ABB RAPID module: 619bfc00.mod

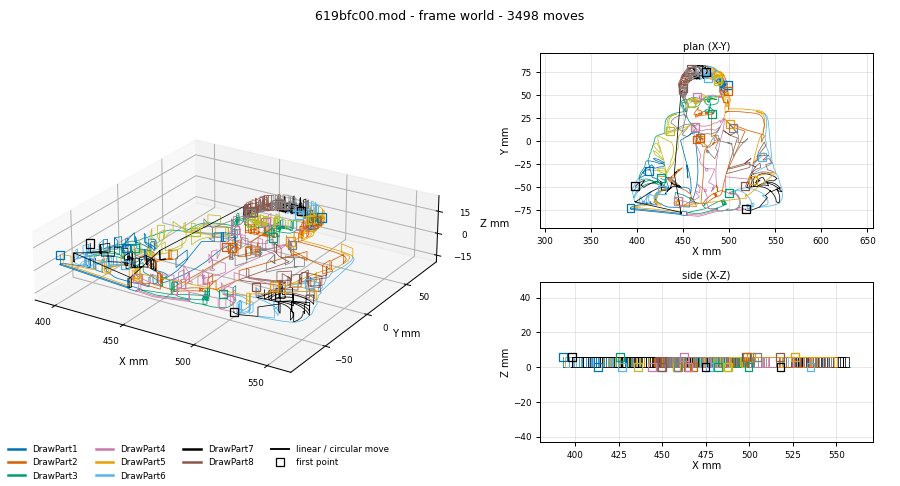
[picture p0: tool path of 619bfc00.mod in frame world, 3498 of 3500 moves have a stored position in this frame; points joined in program order, loops and branches not executed]
MODULE ImageDraw
  ! Generated 2026-10-07 06:22 for ABB GoFa CRB 15000-5/0.95: 344 strokes
  ! Page 250 x 180 mm. Work object wPaper: Z points up, so pen-up is +Z and the tool uses orientation [0,1,0,0].
  PERS tooldata tPen:=[TRUE,[[0,0,120],[1,0,0,0]],[0.3,[0,0,60],[1,0,0,0],0,0,0]];
  PERS wobjdata wPaper:=[FALSE,TRUE,"",[[350,-90,0],[1,0,0,0]],[[0,0,0],[1,0,0,0]]];
  CONST robtarget pOrigin:=[[0,0,0],[0,1,0,0],[0,0,0,0],[9E9,9E9,9E9,9E9,9E9,9E9]];
  CONST jointtarget jHome:=[[0,0,0,0,30,0],[9E9,9E9,9E9,9E9,9E9,9E9]];
  CONST speeddata vTravel:=[250,200,5000,1000];

  PROC DrawImage()
    SingArea\Wrist;
    ConfL\Off;
    ConfJ\Off;
    MoveAbsJ jHome\NoEOffs,vTravel,fine,tPen;
    DrawPart1;
    DrawPart2;
    DrawPart3;
    DrawPart4;
    DrawPart5;
    DrawPart6;
    DrawPart7;
    DrawPart8;
    DrawPart9;
    DrawPart10;
    DrawPart11;
    DrawPart12;
    DrawPart13;
    DrawPart14;
    DrawPart15;
    DrawPart16;
    DrawPart17;
    DrawPart18;
    DrawPart19;
    DrawPart20;
    DrawPart21;
    DrawPart22;
    DrawPart23;
    DrawPart24;
    DrawPart25;
    DrawPart26;
    DrawPart27;
    DrawPart28;
    DrawPart29;
    DrawPart30;
    MoveAbsJ jHome\NoEOffs,vTravel,fine,tPen;
  ENDPROC

  PROC DrawPart1()
    MoveL Offs(pOrigin,42.87,17.43,6.00),vTravel,z5,tPen\WObj:=wPaper;
    MoveL Offs(pOrigin,42.87,17.43,0.00),v60,z0,tPen\WObj:=wPaper;
    MoveL Offs(pOrigin,43.08,16.23,0.00),v40,z0,tPen\WObj:=wPaper;
    MoveL Offs(pOrigin,96.95,10.74,0.00),v40,z0,tPen\WObj:=wPaper;
    MoveL Offs(pOrigin,96.95,10.74,0.00),v40,z0,tPen\WObj:=wPaper;
    MoveL Offs(pOrigin,96.95,12.01,0.00),v40,fine,tPen\WObj:=wPaper;
    MoveL Offs(pOrigin,96.95,12.01,6.00),v60,z5,tPen\WObj:=wPaper;
    MoveL Offs(pOrigin,96.95,10.74,6.00),vTravel,z5,tPen\WObj:=wPaper;
    MoveL Offs(pOrigin,96.95,10.74,0.00),v60,z0,tPen\WObj:=wPaper;
    MoveL Offs(pOrigin,98.22,9.99,0.00),v40,z0,tPen\WObj:=wPaper;
    MoveL Offs(pOrigin,103.43,9.50,0.00),v40,z0,tPen\WObj:=wPaper;
    MoveL Offs(pOrigin,103.54,11.80,0.00),v40,z0,tPen\WObj:=wPaper;
    MoveL Offs(pOrigin,104.39,13.18,0.00),v40,z0,tPen\WObj:=wPaper;
    MoveL Offs(pOrigin,104.39,13.18,0.00),v40,z0,tPen\WObj:=wPaper;
    MoveL Offs(pOrigin,103.96,13.50,0.00),v40,z0,tPen\WObj:=wPaper;
    MoveL Offs(pOrigin,98.44,13.93,0.00),v40,z0,tPen\WObj:=wPaper;
    MoveL Offs(pOrigin,97.27,13.29,0.00),v40,z0,tPen\WObj:=wPaper;
    MoveL Offs(pOrigin,97.27,13.29,0.00),v40,z0,tPen\WObj:=wPaper;
    MoveL Offs(pOrigin,96.91,12.12,0.00),v40,z0,tPen\WObj:=wPaper;
    MoveL Offs(pOrigin,96.10,12.01,0.00),v40,z0,tPen\WObj:=wPaper;
    MoveL Offs(pOrigin,42.87,17.43,0.00),v40,z0,tPen\WObj:=wPaper;
    MoveL Offs(pOrigin,42.87,17.43,0.00),v40,z0,tPen\WObj:=wPaper;
    MoveL Offs(pOrigin,43.08,18.49,0.00),v40,z0,tPen\WObj:=wPaper;
    MoveL Offs(pOrigin,44.04,18.71,0.00),v40,z0,tPen\WObj:=wPaper;
    MoveL Offs(pOrigin,44.04,18.71,0.00),v40,z0,tPen\WObj:=wPaper;
    MoveL Offs(pOrigin,44.36,19.10,0.00),v40,z0,tPen\WObj:=wPaper;
    MoveL Offs(pOrigin,48.29,20.19,0.00),v40,z0,tPen\WObj:=wPaper;
    MoveL Offs(pOrigin,53.81,21.26,0.00),v40,z0,tPen\WObj:=wPaper;
    MoveL Offs(pOrigin,54.66,21.89,0.00),v40,z0,tPen\WObj:=wPaper;
    MoveL Offs(pOrigin,54.66,21.89,0.00),v40,z0,tPen\WObj:=wPaper;
    MoveL Offs(pOrigin,56.36,21.86,0.00),v40,z0,tPen\WObj:=wPaper;
    MoveL Offs(pOrigin,56.26,22.85,0.00),v40,z0,tPen\WObj:=wPaper;
    MoveL Offs(pOrigin,56.26,22.85,0.00),v40,z0,tPen\WObj:=wPaper;
    MoveL Offs(pOrigin,56.19,24.76,0.00),v40,z0,tPen\WObj:=wPaper;
    MoveL Offs(pOrigin,57.11,24.55,0.00),v40,z0,tPen\WObj:=wPaper;
    MoveL Offs(pOrigin,57.11,24.55,0.00),v40,z0,tPen\WObj:=wPaper;
    MoveL Offs(pOrigin,57.74,24.69,0.00),v40,z0,tPen\WObj:=wPaper;
    MoveL Offs(pOrigin,58.17,24.34,0.00),v40,z0,tPen\WObj:=wPaper;
    MoveL Offs(pOrigin,59.12,22.00,0.00),v40,z0,tPen\WObj:=wPaper;
    MoveL Offs(pOrigin,60.61,22.21,0.00),v40,z0,tPen\WObj:=wPaper;
    MoveL Offs(pOrigin,60.51,23.81,0.00),v40,fine,tPen\WObj:=wPaper;
    MoveL Offs(pOrigin,60.51,23.81,6.00),v60,z5,tPen\WObj:=wPaper;
    MoveL Offs(pOrigin,60.72,22.21,6.00),vTravel,z5,tPen\WObj:=wPaper;
    MoveL Offs(pOrigin,60.72,22.21,0.00),v60,z0,tPen\WObj:=wPaper;
    MoveL Offs(pOrigin,61.78,22.42,0.00),v40,fine,tPen\WObj:=wPaper;
    MoveL Offs(pOrigin,61.78,22.42,6.00),v60,z5,tPen\WObj:=wPaper;
    MoveL Offs(pOrigin,63.91,22.64,6.00),vTravel,z5,tPen\WObj:=wPaper;
    MoveL Offs(pOrigin,63.91,22.64,0.00),v60,z0,tPen\WObj:=wPaper;
    MoveL Offs(pOrigin,65.39,22.32,0.00),v40,z0,tPen\WObj:=wPaper;
    MoveL Offs(pOrigin,65.39,22.32,0.00),v40,z0,tPen\WObj:=wPaper;
    MoveL Offs(pOrigin,65.32,23.06,0.00),v40,z0,tPen\WObj:=wPaper;
    MoveL Offs(pOrigin,64.01,24.66,0.00),v40,fine,tPen\WObj:=wPaper;
    MoveL Offs(pOrigin,64.01,24.66,6.00),v60,z5,tPen\WObj:=wPaper;
    MoveL Offs(pOrigin,65.39,22.32,6.00),vTravel,z5,tPen\WObj:=wPaper;
    MoveL Offs(pOrigin,65.39,22.32,0.00),v60,z0,tPen\WObj:=wPaper;
    MoveL Offs(pOrigin,65.82,21.82,0.00),v40,z0,tPen\WObj:=wPaper;
    MoveL Offs(pOrigin,67.09,21.47,0.00),v40,z0,tPen\WObj:=wPaper;
    MoveL Offs(pOrigin,71.34,20.97,0.00),v40,z0,tPen\WObj:=wPaper;
    MoveL Offs(pOrigin,71.27,21.47,0.00),v40,z0,tPen\WObj:=wPaper;
    MoveL Offs(pOrigin,69.43,23.27,0.00),v40,z0,tPen\WObj:=wPaper;
    MoveL Offs(pOrigin,68.47,25.08,0.00),v40,fine,tPen\WObj:=wPaper;
    MoveL Offs(pOrigin,68.47,25.08,6.00),v60,z5,tPen\WObj:=wPaper;
    MoveL Offs(pOrigin,69.86,25.40,6.00),vTravel,z5,tPen\WObj:=wPaper;
    MoveL Offs(pOrigin,69.86,25.40,0.00),v60,z0,tPen\WObj:=wPaper;
    MoveL Offs(pOrigin,69.75,28.06,0.00),v40,z0,tPen\WObj:=wPaper;
    MoveL Offs(pOrigin,69.75,28.06,0.00),v40,z0,tPen\WObj:=wPaper;
    MoveL Offs(pOrigin,70.49,28.02,0.00),v40,z0,tPen\WObj:=wPaper;
    MoveL Offs(pOrigin,70.39,27.21,0.00),v40,z0,tPen\WObj:=wPaper;
    MoveL Offs(pOrigin,70.85,25.51,0.00),v40,z0,tPen\WObj:=wPaper;
    MoveL Offs(pOrigin,71.45,25.29,0.00),v40,z0,tPen\WObj:=wPaper;
    MoveL Offs(pOrigin,71.45,25.29,0.00),v40,z0,tPen\WObj:=wPaper;
    MoveL Offs(pOrigin,72.62,23.59,0.00),v40,z0,tPen\WObj:=wPaper;
    MoveL Offs(pOrigin,74.85,22.81,0.00),v40,z0,tPen\WObj:=wPaper;
    MoveL Offs(pOrigin,75.17,22.32,0.00),v40,z0,tPen\WObj:=wPaper;
    MoveL Offs(pOrigin,75.17,22.32,0.00),v40,z0,tPen\WObj:=wPaper;
    MoveL Offs(pOrigin,76.55,22.14,0.00),v40,z0,tPen\WObj:=wPaper;
    MoveL Offs(pOrigin,77.29,21.29,0.00),v40,z0,tPen\WObj:=wPaper;
    MoveL Offs(pOrigin,81.33,19.31,0.00),v40,z0,tPen\WObj:=wPaper;
    MoveL Offs(pOrigin,84.41,18.60,0.00),v40,z0,tPen\WObj:=wPaper;
    MoveL Offs(pOrigin,94.40,18.39,0.00),v40,z0,tPen\WObj:=wPaper;
    MoveL Offs(pOrigin,97.06,18.60,0.00),v40,z0,tPen\WObj:=wPaper;
    MoveL Offs(pOrigin,99.71,19.34,0.00),v40,z0,tPen\WObj:=wPaper;
    MoveL Offs(pOrigin,99.71,19.34,0.00),v40,z0,tPen\WObj:=wPaper;
    MoveL Offs(pOrigin,100.14,19.02,0.00),v40,z0,tPen\WObj:=wPaper;
    MoveL Offs(pOrigin,106.94,18.71,0.00),v40,fine,tPen\WObj:=wPaper;
    MoveL Offs(pOrigin,106.94,18.71,6.00),v60,z5,tPen\WObj:=wPaper;
    MoveL Offs(pOrigin,106.51,23.59,6.00),vTravel,z5,tPen\WObj:=wPaper;
    MoveL Offs(pOrigin,106.51,23.59,0.00),v60,z0,tPen\WObj:=wPaper;
    MoveL Offs(pOrigin,107.61,24.87,0.00),v40,z0,tPen\WObj:=wPaper;
    MoveL Offs(pOrigin,107.89,26.25,0.00),v40,fine,tPen\WObj:=wPaper;
    MoveL Offs(pOrigin,107.89,26.25,6.00),v60,z5,tPen\WObj:=wPaper;
    MoveL Offs(pOrigin,109.06,27.84,6.00),vTravel,z5,tPen\WObj:=wPaper;
    MoveL Offs(pOrigin,109.06,27.84,0.00),v60,z0,tPen\WObj:=wPaper;
    MoveL Offs(pOrigin,108.00,29.01,0.00),v40,z0,tPen\WObj:=wPaper;
    MoveL Offs(pOrigin,108.53,29.33,0.00),v40,z0,tPen\WObj:=wPaper;
    MoveL Offs(pOrigin,110.12,27.77,0.00),v40,z0,tPen\WObj:=wPaper;
    MoveL Offs(pOrigin,110.66,27.63,0.00),v40,z0,tPen\WObj:=wPaper;
    MoveL Offs(pOrigin,110.66,27.63,0.00),v40,z0,tPen\WObj:=wPaper;
    MoveL Offs(pOrigin,112.14,31.56,0.00),v40,z0,tPen\WObj:=wPaper;
    MoveL Offs(pOrigin,114.27,40.28,0.00),v40,z0,tPen\WObj:=wPaper;
    MoveL Offs(pOrigin,115.01,44.31,0.00),v40,z0,tPen\WObj:=wPaper;
    MoveL Offs(pOrigin,116.07,55.47,0.00),v40,z0,tPen\WObj:=wPaper;
    MoveL Offs(pOrigin,115.86,67.26,0.00),v40,z0,tPen\WObj:=wPaper;
    MoveL Offs(pOrigin,113.74,88.94,0.00),v40,z0,tPen\WObj:=wPaper;
    MoveL Offs(pOrigin,113.74,88.94,0.00),v40,z0,tPen\WObj:=wPaper;
    MoveL Offs(pOrigin,114.27,89.36,0.00),v40,z0,tPen\WObj:=wPaper;
    MoveL Offs(pOrigin,114.48,92.02,0.00),v40,z0,tPen\WObj:=wPaper;
    MoveL Offs(pOrigin,114.48,92.02,0.00),v40,z0,tPen\WObj:=wPaper;
    MoveL Offs(pOrigin,114.91,95.42,0.00),v40,z0,tPen\WObj:=wPaper;
    MoveL Offs(pOrigin,115.76,96.41,0.00),v40,z0,tPen\WObj:=wPaper;
    MoveL Offs(pOrigin,116.29,96.48,0.00),v40,z0,tPen\WObj:=wPaper;
    MoveL Offs(pOrigin,117.24,95.99,0.00),v40,z0,tPen\WObj:=wPaper;
    MoveL Offs(pOrigin,118.73,93.93,0.00),v40,z0,tPen\WObj:=wPaper;
    MoveL Offs(pOrigin,118.52,93.58,0.00),v40,z0,tPen\WObj:=wPaper;
    MoveL Offs(pOrigin,119.09,92.97,0.00),v40,z0,tPen\WObj:=wPaper;
    MoveL Offs(pOrigin,119.47,91.91,0.00),v40,z0,tPen\WObj:=wPaper;
    MoveL Offs(pOrigin,119.26,90.99,0.00),v40,z0,tPen\WObj:=wPaper;
    MoveL Offs(pOrigin,118.52,91.03,0.00),v40,z0,tPen\WObj:=wPaper;
    MoveL Offs(pOrigin,117.85,91.81,0.00),v40,z0,tPen\WObj:=wPaper;
    MoveL Offs(pOrigin,117.56,93.08,0.00),v40,z0,tPen\WObj:=wPaper;
  ENDPROC

  PROC DrawPart2()
    MoveL Offs(pOrigin,117.88,93.54,0.00),v40,z0,tPen\WObj:=wPaper;
    MoveL Offs(pOrigin,118.52,93.58,0.00),v40,z0,tPen\WObj:=wPaper;
    MoveL Offs(pOrigin,118.94,93.08,0.00),v40,z0,tPen\WObj:=wPaper;
    MoveL Offs(pOrigin,118.52,93.51,0.00),v40,z0,tPen\WObj:=wPaper;
    MoveL Offs(pOrigin,118.94,93.08,0.00),v40,fine,tPen\WObj:=wPaper;
    MoveL Offs(pOrigin,118.94,93.08,6.00),v60,z5,tPen\WObj:=wPaper;
    MoveL Offs(pOrigin,120.64,92.97,6.00),vTravel,z5,tPen\WObj:=wPaper;
    MoveL Offs(pOrigin,120.64,92.97,0.00),v60,z0,tPen\WObj:=wPaper;
    MoveL Offs(pOrigin,119.05,95.95,0.00),v40,z0,tPen\WObj:=wPaper;
    MoveL Offs(pOrigin,119.05,95.95,0.00),v40,z0,tPen\WObj:=wPaper;
    MoveL Offs(pOrigin,123.51,94.46,0.00),v40,fine,tPen\WObj:=wPaper;
    MoveL Offs(pOrigin,123.51,94.46,6.00),v60,z5,tPen\WObj:=wPaper;
    MoveL Offs(pOrigin,122.56,92.34,6.00),vTravel,z5,tPen\WObj:=wPaper;
    MoveL Offs(pOrigin,122.56,92.34,0.00),v60,z0,tPen\WObj:=wPaper;
    MoveL Offs(pOrigin,120.64,92.97,0.00),v40,z0,tPen\WObj:=wPaper;
    MoveL Offs(pOrigin,120.64,92.97,0.00),v40,z0,tPen\WObj:=wPaper;
    MoveL Offs(pOrigin,122.41,87.98,0.00),v40,z0,tPen\WObj:=wPaper;
    MoveL Offs(pOrigin,124.68,85.86,0.00),v40,z0,tPen\WObj:=wPaper;
    MoveL Offs(pOrigin,124.89,85.75,0.00),v40,z0,tPen\WObj:=wPaper;
    MoveL Offs(pOrigin,126.49,84.37,0.00),v40,z0,tPen\WObj:=wPaper;
    MoveL Offs(pOrigin,126.49,84.37,0.00),v40,z0,tPen\WObj:=wPaper;
    MoveL Offs(pOrigin,124.47,81.93,0.00),v40,z0,tPen\WObj:=wPaper;
    MoveL Offs(pOrigin,123.58,80.33,0.00),v40,z0,tPen\WObj:=wPaper;
    MoveL Offs(pOrigin,122.66,76.08,0.00),v40,z0,tPen\WObj:=wPaper;
    MoveL Offs(pOrigin,121.71,51.01,0.00),v40,z0,tPen\WObj:=wPaper;
    MoveL Offs(pOrigin,119.37,22.64,0.00),v40,z0,tPen\WObj:=wPaper;
    MoveL Offs(pOrigin,113.21,22.96,0.00),v40,z0,tPen\WObj:=wPaper;
    MoveL Offs(pOrigin,113.21,22.96,0.00),v40,z0,tPen\WObj:=wPaper;
    MoveL Offs(pOrigin,109.06,23.27,0.00),v40,z0,tPen\WObj:=wPaper;
    MoveL Offs(pOrigin,109.06,23.27,0.00),v40,z0,tPen\WObj:=wPaper;
    MoveL Offs(pOrigin,107.26,23.27,0.00),v40,z0,tPen\WObj:=wPaper;
    MoveL Offs(pOrigin,106.51,23.59,0.00),v40,z0,tPen\WObj:=wPaper;
    MoveL Offs(pOrigin,106.51,23.59,0.00),v40,z0,tPen\WObj:=wPaper;
    MoveL Offs(pOrigin,104.92,23.56,0.00),v40,z0,tPen\WObj:=wPaper;
    MoveL Offs(pOrigin,103.64,22.11,0.00),v40,z0,tPen\WObj:=wPaper;
    MoveL Offs(pOrigin,100.67,20.51,0.00),v40,z0,tPen\WObj:=wPaper;
    MoveL Offs(pOrigin,100.67,20.51,0.00),v40,z0,tPen\WObj:=wPaper;
    MoveL Offs(pOrigin,101.09,20.09,0.00),v40,z0,tPen\WObj:=wPaper;
    MoveL Offs(pOrigin,114.48,19.45,0.00),v40,fine,tPen\WObj:=wPaper;
    MoveL Offs(pOrigin,114.48,19.45,6.00),v60,z5,tPen\WObj:=wPaper;
    MoveL Offs(pOrigin,112.99,23.70,6.00),vTravel,z5,tPen\WObj:=wPaper;
    MoveL Offs(pOrigin,112.99,23.70,0.00),v60,z0,tPen\WObj:=wPaper;
    MoveL Offs(pOrigin,112.36,24.76,0.00),v40,z0,tPen\WObj:=wPaper;
    MoveL Offs(pOrigin,112.36,24.76,0.00),v40,z0,tPen\WObj:=wPaper;
    MoveL Offs(pOrigin,110.66,27.63,0.00),v40,fine,tPen\WObj:=wPaper;
    MoveL Offs(pOrigin,110.66,27.63,6.00),v60,z5,tPen\WObj:=wPaper;
    MoveL Offs(pOrigin,110.66,26.36,6.00),vTravel,z5,tPen\WObj:=wPaper;
    MoveL Offs(pOrigin,110.66,26.36,0.00),v60,z0,tPen\WObj:=wPaper;
    MoveL Offs(pOrigin,109.28,27.74,0.00),v40,fine,tPen\WObj:=wPaper;
    MoveL Offs(pOrigin,109.28,27.74,6.00),v60,z5,tPen\WObj:=wPaper;
    MoveL Offs(pOrigin,106.72,28.48,6.00),vTravel,z5,tPen\WObj:=wPaper;
    MoveL Offs(pOrigin,106.72,28.48,0.00),v60,z0,tPen\WObj:=wPaper;
    MoveL Offs(pOrigin,108.53,29.54,0.00),v40,z0,tPen\WObj:=wPaper;
    MoveL Offs(pOrigin,108.74,30.92,0.00),v40,z0,tPen\WObj:=wPaper;
    MoveL Offs(pOrigin,108.00,33.16,0.00),v40,z0,tPen\WObj:=wPaper;
    MoveL Offs(pOrigin,108.00,33.90,0.00),v40,z0,tPen\WObj:=wPaper;
    MoveL Offs(pOrigin,107.89,33.19,0.00),v40,z0,tPen\WObj:=wPaper;
    MoveL Offs(pOrigin,107.15,33.30,0.00),v40,z0,tPen\WObj:=wPaper;
    MoveL Offs(pOrigin,102.58,36.98,0.00),v40,z0,tPen\WObj:=wPaper;
    MoveL Offs(pOrigin,102.58,36.98,0.00),v40,z0,tPen\WObj:=wPaper;
    MoveL Offs(pOrigin,100.24,37.80,0.00),v40,z0,tPen\WObj:=wPaper;
    MoveL Offs(pOrigin,98.33,38.89,0.00),v40,fine,tPen\WObj:=wPaper;
    MoveL Offs(pOrigin,98.33,38.89,6.00),v60,z5,tPen\WObj:=wPaper;
    MoveL Offs(pOrigin,97.80,40.28,6.00),vTravel,z5,tPen\WObj:=wPaper;
    MoveL Offs(pOrigin,97.80,40.28,0.00),v60,z0,tPen\WObj:=wPaper;
    MoveL Offs(pOrigin,95.04,42.22,0.00),v40,z0,tPen\WObj:=wPaper;
    MoveL Offs(pOrigin,94.65,43.14,0.00),v40,z0,tPen\WObj:=wPaper;
    MoveL Offs(pOrigin,94.19,43.36,0.00),v40,z0,tPen\WObj:=wPaper;
    MoveL Offs(pOrigin,94.19,43.36,0.00),v40,z0,tPen\WObj:=wPaper;
    MoveL Offs(pOrigin,91.21,46.33,0.00),v40,z0,tPen\WObj:=wPaper;
    MoveL Offs(pOrigin,90.47,46.86,0.00),v40,z0,tPen\WObj:=wPaper;
    MoveL Offs(pOrigin,90.93,46.47,0.00),v40,z0,tPen\WObj:=wPaper;
    MoveL Offs(pOrigin,86.36,50.37,0.00),v40,z0,tPen\WObj:=wPaper;
    MoveL Offs(pOrigin,95.46,59.72,0.00),v40,fine,tPen\WObj:=wPaper;
    MoveL Offs(pOrigin,95.46,59.72,6.00),v60,z5,tPen\WObj:=wPaper;
    MoveL Offs(pOrigin,94.29,58.66,6.00),vTravel,z5,tPen\WObj:=wPaper;
    MoveL Offs(pOrigin,94.29,58.66,0.00),v60,z0,tPen\WObj:=wPaper;
    MoveL Offs(pOrigin,94.82,59.19,0.00),v40,z0,tPen\WObj:=wPaper;
    MoveL Offs(pOrigin,94.29,58.66,0.00),v40,z0,tPen\WObj:=wPaper;
    MoveL Offs(pOrigin,95.25,58.12,0.00),v40,z0,tPen\WObj:=wPaper;
    MoveL Offs(pOrigin,96.42,59.29,0.00),v40,z0,tPen\WObj:=wPaper;
    MoveL Offs(pOrigin,95.25,58.12,0.00),v40,fine,tPen\WObj:=wPaper;
    MoveL Offs(pOrigin,95.25,58.12,6.00),v60,z5,tPen\WObj:=wPaper;
    MoveL Offs(pOrigin,98.97,61.31,6.00),vTravel,z5,tPen\WObj:=wPaper;
    MoveL Offs(pOrigin,98.97,61.31,0.00),v60,z0,tPen\WObj:=wPaper;
    MoveL Offs(pOrigin,93.66,56.32,0.00),v40,z0,tPen\WObj:=wPaper;
    MoveL Offs(pOrigin,91.18,52.81,0.00),v40,z0,tPen\WObj:=wPaper;
    MoveL Offs(pOrigin,89.62,49.84,0.00),v40,fine,tPen\WObj:=wPaper;
    MoveL Offs(pOrigin,89.62,49.84,6.00),v60,z5,tPen\WObj:=wPaper;
    MoveL Offs(pOrigin,87.07,51.33,6.00),vTravel,z5,tPen\WObj:=wPaper;
    MoveL Offs(pOrigin,87.07,51.33,0.00),v60,z0,tPen\WObj:=wPaper;
    MoveL Offs(pOrigin,87.49,51.75,0.00),v40,z0,tPen\WObj:=wPaper;
    MoveL Offs(pOrigin,87.07,51.33,0.00),v40,z0,tPen\WObj:=wPaper;
    MoveL Offs(pOrigin,86.32,50.47,0.00),v40,z0,tPen\WObj:=wPaper;
    MoveL Offs(pOrigin,84.84,50.79,0.00),v40,z0,tPen\WObj:=wPaper;
    MoveL Offs(pOrigin,84.84,50.79,0.00),v40,z0,tPen\WObj:=wPaper;
    MoveL Offs(pOrigin,83.24,49.20,0.00),v40,z0,tPen\WObj:=wPaper;
    MoveL Offs(pOrigin,83.24,49.20,0.00),v40,z0,tPen\WObj:=wPaper;
    MoveL Offs(pOrigin,83.99,48.03,0.00),v40,z0,tPen\WObj:=wPaper;
    MoveL Offs(pOrigin,90.36,42.22,0.00),v40,z0,tPen\WObj:=wPaper;
    MoveL Offs(pOrigin,90.79,41.48,0.00),v40,z0,tPen\WObj:=wPaper;
    MoveL Offs(pOrigin,93.09,41.02,0.00),v40,z0,tPen\WObj:=wPaper;
    MoveL Offs(pOrigin,93.09,41.55,0.00),v40,z0,tPen\WObj:=wPaper;
    MoveL Offs(pOrigin,88.45,45.69,0.00),v40,z0,tPen\WObj:=wPaper;
    MoveL Offs(pOrigin,87.92,46.01,0.00),v40,z0,tPen\WObj:=wPaper;
    MoveL Offs(pOrigin,88.17,45.84,0.00),v40,z0,tPen\WObj:=wPaper;
    MoveL Offs(pOrigin,84.62,48.88,0.00),v40,fine,tPen\WObj:=wPaper;
    MoveL Offs(pOrigin,84.62,48.88,6.00),v60,z5,tPen\WObj:=wPaper;
    MoveL Offs(pOrigin,83.24,49.20,6.00),vTravel,z5,tPen\WObj:=wPaper;
    MoveL Offs(pOrigin,83.24,49.20,0.00),v60,z0,tPen\WObj:=wPaper;
    MoveL Offs(pOrigin,82.89,49.52,0.00),v40,z0,tPen\WObj:=wPaper;
    MoveL Offs(pOrigin,82.82,50.26,0.00),v40,z0,tPen\WObj:=wPaper;
    MoveL Offs(pOrigin,82.82,50.26,0.00),v40,z0,tPen\WObj:=wPaper;
    MoveL Offs(pOrigin,81.83,51.11,0.00),v40,z0,tPen\WObj:=wPaper;
    MoveL Offs(pOrigin,81.44,53.45,0.00),v40,z0,tPen\WObj:=wPaper;
    MoveL Offs(pOrigin,81.44,53.45,0.00),v40,z0,tPen\WObj:=wPaper;
    MoveL Offs(pOrigin,80.27,52.25,0.00),v40,z0,tPen\WObj:=wPaper;
    MoveL Offs(pOrigin,78.99,51.96,0.00),v40,z0,tPen\WObj:=wPaper;
    MoveL Offs(pOrigin,73.26,52.28,0.00),v40,fine,tPen\WObj:=wPaper;
    MoveL Offs(pOrigin,73.26,52.28,6.00),v60,z5,tPen\WObj:=wPaper;
  ENDPROC

  PROC DrawPart3()
    MoveL Offs(pOrigin,75.70,49.84,6.00),vTravel,z5,tPen\WObj:=wPaper;
    MoveL Offs(pOrigin,75.70,49.84,0.00),v60,z0,tPen\WObj:=wPaper;
    MoveL Offs(pOrigin,79.10,48.14,0.00),v40,z0,tPen\WObj:=wPaper;
    MoveL Offs(pOrigin,80.48,48.67,0.00),v40,z0,tPen\WObj:=wPaper;
    MoveL Offs(pOrigin,80.48,48.67,0.00),v40,z0,tPen\WObj:=wPaper;
    MoveL Offs(pOrigin,80.38,44.53,0.00),v40,z0,tPen\WObj:=wPaper;
    MoveL Offs(pOrigin,79.21,41.12,0.00),v40,z0,tPen\WObj:=wPaper;
    MoveL Offs(pOrigin,75.06,42.36,0.00),v40,z0,tPen\WObj:=wPaper;
    MoveL Offs(pOrigin,72.41,43.53,0.00),v40,z0,tPen\WObj:=wPaper;
    MoveL Offs(pOrigin,69.01,46.15,0.00),v40,z0,tPen\WObj:=wPaper;
    MoveL Offs(pOrigin,65.39,47.71,0.00),v40,z0,tPen\WObj:=wPaper;
    MoveL Offs(pOrigin,65.39,47.71,0.00),v40,z0,tPen\WObj:=wPaper;
    MoveL Offs(pOrigin,65.07,47.29,0.00),v40,z0,tPen\WObj:=wPaper;
    MoveL Offs(pOrigin,62.42,47.39,0.00),v40,z0,tPen\WObj:=wPaper;
    MoveL Offs(pOrigin,60.40,46.90,0.00),v40,z0,tPen\WObj:=wPaper;
    MoveL Offs(pOrigin,58.06,45.84,0.00),v40,z0,tPen\WObj:=wPaper;
    MoveL Offs(pOrigin,55.94,44.31,0.00),v40,z0,tPen\WObj:=wPaper;
    MoveL Offs(pOrigin,52.29,39.96,0.00),v40,z0,tPen\WObj:=wPaper;
    MoveL Offs(pOrigin,50.59,36.77,0.00),v40,z0,tPen\WObj:=wPaper;
    MoveL Offs(pOrigin,49.99,34.86,0.00),v40,z0,tPen\WObj:=wPaper;
    MoveL Offs(pOrigin,49.99,34.86,0.00),v40,z0,tPen\WObj:=wPaper;
    MoveL Offs(pOrigin,51.90,36.34,0.00),v40,z0,tPen\WObj:=wPaper;
    MoveL Offs(pOrigin,55.94,41.02,0.00),v40,z0,tPen\WObj:=wPaper;
    MoveL Offs(pOrigin,57.74,42.44,0.00),v40,z0,tPen\WObj:=wPaper;
    MoveL Offs(pOrigin,61.25,43.89,0.00),v40,z0,tPen\WObj:=wPaper;
    MoveL Offs(pOrigin,64.12,44.21,0.00),v40,z0,tPen\WObj:=wPaper;
    MoveL Offs(pOrigin,64.12,44.21,0.00),v40,z0,tPen\WObj:=wPaper;
    MoveL Offs(pOrigin,67.09,44.31,0.00),v40,z0,tPen\WObj:=wPaper;
    MoveL Offs(pOrigin,71.77,43.78,0.00),v40,fine,tPen\WObj:=wPaper;
    MoveL Offs(pOrigin,71.77,43.78,6.00),v60,z5,tPen\WObj:=wPaper;
    MoveL Offs(pOrigin,69.86,45.27,6.00),vTravel,z5,tPen\WObj:=wPaper;
    MoveL Offs(pOrigin,69.86,45.27,0.00),v60,z0,tPen\WObj:=wPaper;
    MoveL Offs(pOrigin,69.32,45.16,0.00),v40,z0,tPen\WObj:=wPaper;
    MoveL Offs(pOrigin,67.94,45.87,0.00),v40,z0,tPen\WObj:=wPaper;
    MoveL Offs(pOrigin,67.62,46.65,0.00),v40,fine,tPen\WObj:=wPaper;
    MoveL Offs(pOrigin,67.62,46.65,6.00),v60,z5,tPen\WObj:=wPaper;
    MoveL Offs(pOrigin,65.39,47.71,6.00),vTravel,z5,tPen\WObj:=wPaper;
    MoveL Offs(pOrigin,65.39,47.71,0.00),v60,z0,tPen\WObj:=wPaper;
    MoveL Offs(pOrigin,63.91,48.46,0.00),v40,z0,tPen\WObj:=wPaper;
    MoveL Offs(pOrigin,60.51,49.20,0.00),v40,z0,tPen\WObj:=wPaper;
    MoveL Offs(pOrigin,56.26,48.99,0.00),v40,z0,tPen\WObj:=wPaper;
    MoveL Offs(pOrigin,53.07,47.92,0.00),v40,fine,tPen\WObj:=wPaper;
    MoveL Offs(pOrigin,53.07,47.92,6.00),v60,z5,tPen\WObj:=wPaper;
    MoveL Offs(pOrigin,52.01,49.84,6.00),vTravel,z5,tPen\WObj:=wPaper;
    MoveL Offs(pOrigin,52.01,49.84,0.00),v60,z0,tPen\WObj:=wPaper;
    MoveL Offs(pOrigin,52.86,53.34,0.00),v40,z0,tPen\WObj:=wPaper;
    MoveL Offs(pOrigin,54.10,56.53,0.00),v40,z0,tPen\WObj:=wPaper;
    MoveL Offs(pOrigin,58.10,61.95,0.00),v40,z0,tPen\WObj:=wPaper;
    MoveL Offs(pOrigin,59.41,67.69,0.00),v40,z0,tPen\WObj:=wPaper;
    MoveL Offs(pOrigin,60.51,68.79,0.00),v40,z0,tPen\WObj:=wPaper;
    MoveL Offs(pOrigin,61.89,69.07,0.00),v40,z0,tPen\WObj:=wPaper;
    MoveL Offs(pOrigin,61.89,69.07,0.00),v40,z0,tPen\WObj:=wPaper;
    MoveL Offs(pOrigin,62.03,70.56,0.00),v40,z0,tPen\WObj:=wPaper;
    MoveL Offs(pOrigin,63.48,72.79,0.00),v40,z0,tPen\WObj:=wPaper;
    MoveL Offs(pOrigin,63.66,76.19,0.00),v40,z0,tPen\WObj:=wPaper;
    MoveL Offs(pOrigin,64.90,77.68,0.00),v40,z0,tPen\WObj:=wPaper;
    MoveL Offs(pOrigin,65.18,78.53,0.00),v40,z0,tPen\WObj:=wPaper;
    MoveL Offs(pOrigin,65.25,81.18,0.00),v40,z0,tPen\WObj:=wPaper;
    MoveL Offs(pOrigin,66.78,82.99,0.00),v40,z0,tPen\WObj:=wPaper;
    MoveL Offs(pOrigin,66.88,85.43,0.00),v40,z0,tPen\WObj:=wPaper;
    MoveL Offs(pOrigin,67.59,86.39,0.00),v40,z0,tPen\WObj:=wPaper;
    MoveL Offs(pOrigin,68.47,89.15,0.00),v40,z0,tPen\WObj:=wPaper;
    MoveL Offs(pOrigin,69.50,93.72,0.00),v40,z0,tPen\WObj:=wPaper;
    MoveL Offs(pOrigin,71.03,95.84,0.00),v40,z0,tPen\WObj:=wPaper;
    MoveL Offs(pOrigin,72.51,96.38,0.00),v40,z0,tPen\WObj:=wPaper;
    MoveL Offs(pOrigin,72.51,96.38,0.00),v40,z0,tPen\WObj:=wPaper;
    MoveL Offs(pOrigin,75.06,97.44,0.00),v40,z0,tPen\WObj:=wPaper;
    MoveL Offs(pOrigin,79.84,98.78,0.00),v40,z0,tPen\WObj:=wPaper;
    MoveL Offs(pOrigin,80.16,99.14,0.00),v40,z0,tPen\WObj:=wPaper;
    MoveL Offs(pOrigin,80.16,99.14,0.00),v40,z0,tPen\WObj:=wPaper;
    MoveL Offs(pOrigin,80.16,105.83,0.00),v40,z0,tPen\WObj:=wPaper;
    MoveL Offs(pOrigin,80.59,110.82,0.00),v40,z0,tPen\WObj:=wPaper;
    MoveL Offs(pOrigin,81.40,113.59,0.00),v40,z0,tPen\WObj:=wPaper;
    MoveL Offs(pOrigin,82.93,116.03,0.00),v40,z0,tPen\WObj:=wPaper;
    MoveL Offs(pOrigin,85.37,118.09,0.00),v40,z0,tPen\WObj:=wPaper;
    MoveL Offs(pOrigin,89.30,119.89,0.00),v40,z0,tPen\WObj:=wPaper;
    MoveL Offs(pOrigin,93.02,120.92,0.00),v40,z0,tPen\WObj:=wPaper;
    MoveL Offs(pOrigin,100.88,122.30,0.00),v40,z0,tPen\WObj:=wPaper;
    MoveL Offs(pOrigin,100.88,122.30,0.00),v40,z0,tPen\WObj:=wPaper;
    MoveL Offs(pOrigin,100.17,124.85,0.00),v40,z0,tPen\WObj:=wPaper;
    MoveL Offs(pOrigin,98.37,127.82,0.00),v40,z0,tPen\WObj:=wPaper;
    MoveL Offs(pOrigin,97.69,130.06,0.00),v40,z0,tPen\WObj:=wPaper;
    MoveL Offs(pOrigin,98.08,133.03,0.00),v40,z0,tPen\WObj:=wPaper;
    MoveL Offs(pOrigin,98.86,134.09,0.00),v40,z0,tPen\WObj:=wPaper;
    MoveL Offs(pOrigin,100.03,134.73,0.00),v40,z0,tPen\WObj:=wPaper;
    MoveL Offs(pOrigin,100.14,135.48,0.00),v40,z0,tPen\WObj:=wPaper;
    MoveL Offs(pOrigin,100.14,134.73,0.00),v40,z0,tPen\WObj:=wPaper;
    MoveL Offs(pOrigin,101.41,134.41,0.00),v40,z0,tPen\WObj:=wPaper;
    MoveL Offs(pOrigin,101.41,134.41,0.00),v40,z0,tPen\WObj:=wPaper;
    MoveL Offs(pOrigin,101.55,133.14,0.00),v40,z0,tPen\WObj:=wPaper;
    MoveL Offs(pOrigin,102.05,132.61,0.00),v40,z0,tPen\WObj:=wPaper;
    MoveL Offs(pOrigin,102.58,132.18,0.00),v40,z0,tPen\WObj:=wPaper;
    MoveL Offs(pOrigin,102.37,131.44,0.00),v40,z0,tPen\WObj:=wPaper;
    MoveL Offs(pOrigin,100.56,132.36,0.00),v40,z0,tPen\WObj:=wPaper;
    MoveL Offs(pOrigin,99.54,132.39,0.00),v40,z0,tPen\WObj:=wPaper;
    MoveL Offs(pOrigin,99.07,129.84,0.00),v40,z0,tPen\WObj:=wPaper;
    MoveL Offs(pOrigin,100.03,127.61,0.00),v40,fine,tPen\WObj:=wPaper;
    MoveL Offs(pOrigin,100.03,127.61,6.00),v60,z5,tPen\WObj:=wPaper;
    MoveL Offs(pOrigin,100.67,129.21,6.00),vTravel,z5,tPen\WObj:=wPaper;
    MoveL Offs(pOrigin,100.67,129.21,0.00),v60,z0,tPen\WObj:=wPaper;
    MoveL Offs(pOrigin,100.78,126.44,0.00),v40,z0,tPen\WObj:=wPaper;
    MoveL Offs(pOrigin,102.47,122.30,0.00),v40,z0,tPen\WObj:=wPaper;
    MoveL Offs(pOrigin,103.32,122.62,0.00),v40,z0,tPen\WObj:=wPaper;
    MoveL Offs(pOrigin,103.22,123.68,0.00),v40,fine,tPen\WObj:=wPaper;
    MoveL Offs(pOrigin,103.22,123.68,6.00),v60,z5,tPen\WObj:=wPaper;
    MoveL Offs(pOrigin,103.54,121.13,6.00),vTravel,z5,tPen\WObj:=wPaper;
    MoveL Offs(pOrigin,103.54,121.13,0.00),v60,z0,tPen\WObj:=wPaper;
    MoveL Offs(pOrigin,104.18,116.35,0.00),v40,z0,tPen\WObj:=wPaper;
    MoveL Offs(pOrigin,104.18,116.35,0.00),v40,z0,tPen\WObj:=wPaper;
    MoveL Offs(pOrigin,106.19,112.31,0.00),v40,z0,tPen\WObj:=wPaper;
    MoveL Offs(pOrigin,108.64,109.27,0.00),v40,z0,tPen\WObj:=wPaper;
    MoveL Offs(pOrigin,110.02,108.49,0.00),v40,z0,tPen\WObj:=wPaper;
    MoveL Offs(pOrigin,110.02,108.49,0.00),v40,z0,tPen\WObj:=wPaper;
    MoveL Offs(pOrigin,113.31,107.11,0.00),v40,fine,tPen\WObj:=wPaper;
    MoveL Offs(pOrigin,113.31,107.11,6.00),v60,z5,tPen\WObj:=wPaper;
    MoveL Offs(pOrigin,111.72,106.26,6.00),vTravel,z5,tPen\WObj:=wPaper;
    MoveL Offs(pOrigin,111.72,106.26,0.00),v60,z0,tPen\WObj:=wPaper;
    MoveL Offs(pOrigin,110.97,107.00,0.00),v40,z0,tPen\WObj:=wPaper;
    MoveL Offs(pOrigin,111.72,106.26,0.00),v40,fine,tPen\WObj:=wPaper;
    MoveL Offs(pOrigin,111.72,106.26,6.00),v60,z5,tPen\WObj:=wPaper;
  ENDPROC

  PROC DrawPart4()
    MoveL Offs(pOrigin,112.68,105.30,6.00),vTravel,z5,tPen\WObj:=wPaper;
    MoveL Offs(pOrigin,112.68,105.30,0.00),v60,z0,tPen\WObj:=wPaper;
    MoveL Offs(pOrigin,111.82,106.15,0.00),v40,z0,tPen\WObj:=wPaper;
    MoveL Offs(pOrigin,112.68,105.30,0.00),v40,fine,tPen\WObj:=wPaper;
    MoveL Offs(pOrigin,112.68,105.30,6.00),v60,z5,tPen\WObj:=wPaper;
    MoveL Offs(pOrigin,113.53,104.34,6.00),vTravel,z5,tPen\WObj:=wPaper;
    MoveL Offs(pOrigin,113.53,104.34,0.00),v60,z0,tPen\WObj:=wPaper;
    MoveL Offs(pOrigin,110.83,107.28,0.00),v40,z0,tPen\WObj:=wPaper;
    MoveL Offs(pOrigin,110.27,107.53,0.00),v40,z0,tPen\WObj:=wPaper;
    MoveL Offs(pOrigin,110.02,108.49,0.00),v40,z0,tPen\WObj:=wPaper;
    MoveL Offs(pOrigin,110.23,107.43,0.00),v40,z0,tPen\WObj:=wPaper;
    MoveL Offs(pOrigin,111.19,100.41,0.00),v40,z0,tPen\WObj:=wPaper;
    MoveL Offs(pOrigin,111.19,100.41,0.00),v40,z0,tPen\WObj:=wPaper;
    MoveL Offs(pOrigin,112.46,95.42,0.00),v40,z0,tPen\WObj:=wPaper;
    MoveL Offs(pOrigin,113.42,89.26,0.00),v40,z0,tPen\WObj:=wPaper;
    MoveL Offs(pOrigin,113.74,88.94,0.00),v40,fine,tPen\WObj:=wPaper;
    MoveL Offs(pOrigin,113.74,88.94,6.00),v60,z5,tPen\WObj:=wPaper;
    MoveL Offs(pOrigin,114.06,86.28,6.00),vTravel,z5,tPen\WObj:=wPaper;
    MoveL Offs(pOrigin,114.06,86.28,0.00),v60,z0,tPen\WObj:=wPaper;
    MoveL Offs(pOrigin,114.66,85.86,0.00),v40,z0,tPen\WObj:=wPaper;
    MoveL Offs(pOrigin,119.37,74.28,0.00),v40,fine,tPen\WObj:=wPaper;
    MoveL Offs(pOrigin,119.37,74.28,6.00),v60,z5,tPen\WObj:=wPaper;
    MoveL Offs(pOrigin,117.78,70.34,6.00),vTravel,z5,tPen\WObj:=wPaper;
    MoveL Offs(pOrigin,117.78,70.34,0.00),v60,z0,tPen\WObj:=wPaper;
    MoveL Offs(pOrigin,118.62,66.31,0.00),v40,fine,tPen\WObj:=wPaper;
    MoveL Offs(pOrigin,118.62,66.31,6.00),v60,z5,tPen\WObj:=wPaper;
    MoveL Offs(pOrigin,124.86,60.39,6.00),vTravel,z5,tPen\WObj:=wPaper;
    MoveL Offs(pOrigin,124.86,60.39,0.00),v60,z0,tPen\WObj:=wPaper;
    MoveL Offs(pOrigin,125.85,60.57,0.00),v40,z0,tPen\WObj:=wPaper;
    MoveL Offs(pOrigin,126.59,60.14,0.00),v40,z0,tPen\WObj:=wPaper;
    MoveL Offs(pOrigin,127.02,59.08,0.00),v40,z0,tPen\WObj:=wPaper;
    MoveL Offs(pOrigin,126.59,58.02,0.00),v40,z0,tPen\WObj:=wPaper;
    MoveL Offs(pOrigin,125.21,57.70,0.00),v40,z0,tPen\WObj:=wPaper;
    MoveL Offs(pOrigin,124.47,58.12,0.00),v40,z0,tPen\WObj:=wPaper;
    MoveL Offs(pOrigin,124.15,59.51,0.00),v40,z0,tPen\WObj:=wPaper;
    MoveL Offs(pOrigin,124.86,60.39,0.00),v40,fine,tPen\WObj:=wPaper;
    MoveL Offs(pOrigin,124.86,60.39,6.00),v60,z5,tPen\WObj:=wPaper;
    MoveL Offs(pOrigin,134.35,60.04,6.00),vTravel,z5,tPen\WObj:=wPaper;
    MoveL Offs(pOrigin,134.35,60.04,0.00),v60,z0,tPen\WObj:=wPaper;
    MoveL Offs(pOrigin,131.09,52.17,0.00),v40,z0,tPen\WObj:=wPaper;
    MoveL Offs(pOrigin,127.55,45.48,0.00),v40,fine,tPen\WObj:=wPaper;
    MoveL Offs(pOrigin,127.55,45.48,6.00),v60,z5,tPen\WObj:=wPaper;
    MoveL Offs(pOrigin,133.93,42.19,6.00),vTravel,z5,tPen\WObj:=wPaper;
    MoveL Offs(pOrigin,133.93,42.19,0.00),v60,z0,tPen\WObj:=wPaper;
    MoveL Offs(pOrigin,131.69,39.32,0.00),v40,fine,tPen\WObj:=wPaper;
    MoveL Offs(pOrigin,131.69,39.32,6.00),v60,z5,tPen\WObj:=wPaper;
    MoveL Offs(pOrigin,132.65,38.26,6.00),vTravel,z5,tPen\WObj:=wPaper;
    MoveL Offs(pOrigin,132.65,38.26,0.00),v60,z0,tPen\WObj:=wPaper;
    MoveL Offs(pOrigin,132.97,38.58,0.00),v40,z0,tPen\WObj:=wPaper;
    MoveL Offs(pOrigin,132.65,38.26,0.00),v40,z0,tPen\WObj:=wPaper;
    MoveL Offs(pOrigin,133.29,39.00,0.00),v40,z0,tPen\WObj:=wPaper;
    MoveL Offs(pOrigin,133.61,39.32,0.00),v40,z0,tPen\WObj:=wPaper;
    MoveL Offs(pOrigin,133.29,39.00,0.00),v40,fine,tPen\WObj:=wPaper;
    MoveL Offs(pOrigin,133.29,39.00,6.00),v60,z5,tPen\WObj:=wPaper;
    MoveL Offs(pOrigin,130.42,35.81,6.00),vTravel,z5,tPen\WObj:=wPaper;
    MoveL Offs(pOrigin,130.42,35.81,0.00),v60,z0,tPen\WObj:=wPaper;
    MoveL Offs(pOrigin,136.37,42.72,0.00),v40,z0,tPen\WObj:=wPaper;
    MoveL Offs(pOrigin,136.37,42.72,0.00),v40,z0,tPen\WObj:=wPaper;
    MoveL Offs(pOrigin,135.62,51.22,0.00),v40,z0,tPen\WObj:=wPaper;
    MoveL Offs(pOrigin,135.62,59.83,0.00),v40,z0,tPen\WObj:=wPaper;
    MoveL Offs(pOrigin,136.48,69.28,0.00),v40,z0,tPen\WObj:=wPaper;
    MoveL Offs(pOrigin,137.86,78.84,0.00),v40,z0,tPen\WObj:=wPaper;
    MoveL Offs(pOrigin,137.86,78.84,0.00),v40,z0,tPen\WObj:=wPaper;
    MoveL Offs(pOrigin,140.19,90.21,0.00),v40,z0,tPen\WObj:=wPaper;
    MoveL Offs(pOrigin,143.38,102.01,0.00),v40,z0,tPen\WObj:=wPaper;
    MoveL Offs(pOrigin,143.38,102.01,0.00),v40,z0,tPen\WObj:=wPaper;
    MoveL Offs(pOrigin,144.55,109.23,0.00),v40,z0,tPen\WObj:=wPaper;
    MoveL Offs(pOrigin,144.55,113.16,0.00),v40,z0,tPen\WObj:=wPaper;
    MoveL Offs(pOrigin,144.12,113.91,0.00),v40,z0,tPen\WObj:=wPaper;
    MoveL Offs(pOrigin,144.02,114.76,0.00),v40,z0,tPen\WObj:=wPaper;
    MoveL Offs(pOrigin,143.27,114.33,0.00),v40,z0,tPen\WObj:=wPaper;
    MoveL Offs(pOrigin,140.51,110.40,0.00),v40,fine,tPen\WObj:=wPaper;
    MoveL Offs(pOrigin,140.51,110.40,6.00),v60,z5,tPen\WObj:=wPaper;
    MoveL Offs(pOrigin,140.19,113.06,6.00),vTravel,z5,tPen\WObj:=wPaper;
    MoveL Offs(pOrigin,140.19,113.06,0.00),v60,z0,tPen\WObj:=wPaper;
    MoveL Offs(pOrigin,136.90,110.08,0.00),v40,fine,tPen\WObj:=wPaper;
    MoveL Offs(pOrigin,136.90,110.08,6.00),v60,z5,tPen\WObj:=wPaper;
    MoveL Offs(pOrigin,133.61,109.97,6.00),vTravel,z5,tPen\WObj:=wPaper;
    MoveL Offs(pOrigin,133.61,109.97,0.00),v60,z0,tPen\WObj:=wPaper;
    MoveL Offs(pOrigin,130.21,107.81,0.00),v40,z0,tPen\WObj:=wPaper;
    MoveL Offs(pOrigin,127.23,107.00,0.00),v40,z0,tPen\WObj:=wPaper;
    MoveL Offs(pOrigin,123.51,106.47,0.00),v40,z0,tPen\WObj:=wPaper;
    MoveL Offs(pOrigin,118.84,106.79,0.00),v40,z0,tPen\WObj:=wPaper;
    MoveL Offs(pOrigin,116.61,107.71,0.00),v40,z0,tPen\WObj:=wPaper;
    MoveL Offs(pOrigin,114.59,109.02,0.00),v40,fine,tPen\WObj:=wPaper;
    MoveL Offs(pOrigin,114.59,109.02,6.00),v60,z5,tPen\WObj:=wPaper;
    MoveL Offs(pOrigin,113.53,104.34,6.00),vTravel,z5,tPen\WObj:=wPaper;
    MoveL Offs(pOrigin,113.53,104.34,0.00),v60,z0,tPen\WObj:=wPaper;
    MoveL Offs(pOrigin,117.03,102.40,0.00),v40,z0,tPen\WObj:=wPaper;
    MoveL Offs(pOrigin,119.69,101.37,0.00),v40,fine,tPen\WObj:=wPaper;
    MoveL Offs(pOrigin,119.69,101.37,6.00),v60,z5,tPen\WObj:=wPaper;
    MoveL Offs(pOrigin,122.45,101.90,6.00),vTravel,z5,tPen\WObj:=wPaper;
    MoveL Offs(pOrigin,122.45,101.90,0.00),v60,z0,tPen\WObj:=wPaper;
    MoveL Offs(pOrigin,125.53,103.07,0.00),v40,z0,tPen\WObj:=wPaper;
    MoveL Offs(pOrigin,129.14,102.75,0.00),v40,z0,tPen\WObj:=wPaper;
    MoveL Offs(pOrigin,131.06,102.96,0.00),v40,fine,tPen\WObj:=wPaper;
    MoveL Offs(pOrigin,131.06,102.96,6.00),v60,z5,tPen\WObj:=wPaper;
    MoveL Offs(pOrigin,134.88,102.11,6.00),vTravel,z5,tPen\WObj:=wPaper;
    MoveL Offs(pOrigin,134.88,102.11,0.00),v60,z0,tPen\WObj:=wPaper;
    MoveL Offs(pOrigin,140.19,105.83,0.00),v40,z0,tPen\WObj:=wPaper;
    MoveL Offs(pOrigin,140.19,105.83,0.00),v40,z0,tPen\WObj:=wPaper;
    MoveL Offs(pOrigin,142.99,111.25,0.00),v40,z0,tPen\WObj:=wPaper;
    MoveL Offs(pOrigin,144.12,114.12,0.00),v40,z0,tPen\WObj:=wPaper;
    MoveL Offs(pOrigin,144.12,115.07,0.00),v40,fine,tPen\WObj:=wPaper;
    MoveL Offs(pOrigin,144.12,115.07,6.00),v60,z5,tPen\WObj:=wPaper;
    MoveL Offs(pOrigin,148.06,111.14,6.00),vTravel,z5,tPen\WObj:=wPaper;
    MoveL Offs(pOrigin,148.06,111.14,0.00),v60,z0,tPen\WObj:=wPaper;
    MoveL Offs(pOrigin,147.21,111.99,0.00),v40,z0,tPen\WObj:=wPaper;
    MoveL Offs(pOrigin,148.06,111.14,0.00),v40,fine,tPen\WObj:=wPaper;
    MoveL Offs(pOrigin,148.06,111.14,6.00),v60,z5,tPen\WObj:=wPaper;
    MoveL Offs(pOrigin,148.91,110.29,6.00),vTravel,z5,tPen\WObj:=wPaper;
    MoveL Offs(pOrigin,148.91,110.29,0.00),v60,z0,tPen\WObj:=wPaper;
    MoveL Offs(pOrigin,148.16,111.04,0.00),v40,z0,tPen\WObj:=wPaper;
    MoveL Offs(pOrigin,148.91,110.29,0.00),v40,fine,tPen\WObj:=wPaper;
    MoveL Offs(pOrigin,148.91,110.29,6.00),v60,z5,tPen\WObj:=wPaper;
    MoveL Offs(pOrigin,149.86,109.34,6.00),vTravel,z5,tPen\WObj:=wPaper;
    MoveL Offs(pOrigin,149.86,109.34,0.00),v60,z0,tPen\WObj:=wPaper;
    MoveL Offs(pOrigin,149.01,110.19,0.00),v40,z0,tPen\WObj:=wPaper;
    MoveL Offs(pOrigin,149.86,109.34,0.00),v40,fine,tPen\WObj:=wPaper;
    MoveL Offs(pOrigin,149.86,109.34,6.00),v60,z5,tPen\WObj:=wPaper;
  ENDPROC

  PROC DrawPart5()
    MoveL Offs(pOrigin,151.03,108.70,6.00),vTravel,z5,tPen\WObj:=wPaper;
    MoveL Offs(pOrigin,151.03,108.70,0.00),v60,z0,tPen\WObj:=wPaper;
    MoveL Offs(pOrigin,150.18,109.12,0.00),v40,z0,tPen\WObj:=wPaper;
    MoveL Offs(pOrigin,145.29,114.44,0.00),v40,z0,tPen\WObj:=wPaper;
    MoveL Offs(pOrigin,144.16,115.18,0.00),v40,z0,tPen\WObj:=wPaper;
    MoveL Offs(pOrigin,145.40,119.32,0.00),v40,z0,tPen\WObj:=wPaper;
    MoveL Offs(pOrigin,145.72,121.77,0.00),v40,z0,tPen\WObj:=wPaper;
    MoveL Offs(pOrigin,145.72,121.77,0.00),v40,z0,tPen\WObj:=wPaper;
    MoveL Offs(pOrigin,145.29,126.34,0.00),v40,z0,tPen\WObj:=wPaper;
    MoveL Offs(pOrigin,145.40,127.51,0.00),v40,z0,tPen\WObj:=wPaper;
    MoveL Offs(pOrigin,145.93,128.57,0.00),v40,z0,tPen\WObj:=wPaper;
    MoveL Offs(pOrigin,145.93,128.57,0.00),v40,z0,tPen\WObj:=wPaper;
    MoveL Offs(pOrigin,146.14,130.59,0.00),v40,z0,tPen\WObj:=wPaper;
    MoveL Offs(pOrigin,144.87,132.82,0.00),v40,z0,tPen\WObj:=wPaper;
    MoveL Offs(pOrigin,145.40,132.93,0.00),v40,z0,tPen\WObj:=wPaper;
    MoveL Offs(pOrigin,146.46,131.54,0.00),v40,fine,tPen\WObj:=wPaper;
    MoveL Offs(pOrigin,146.46,131.54,6.00),v60,z5,tPen\WObj:=wPaper;
    MoveL Offs(pOrigin,147.42,130.69,6.00),vTravel,z5,tPen\WObj:=wPaper;
    MoveL Offs(pOrigin,147.42,130.69,0.00),v60,z0,tPen\WObj:=wPaper;
    MoveL Offs(pOrigin,146.89,129.21,0.00),v40,z0,tPen\WObj:=wPaper;
    MoveL Offs(pOrigin,145.93,128.57,0.00),v40,fine,tPen\WObj:=wPaper;
    MoveL Offs(pOrigin,145.93,128.57,6.00),v60,z5,tPen\WObj:=wPaper;
    MoveL Offs(pOrigin,147.63,127.40,6.00),vTravel,z5,tPen\WObj:=wPaper;
    MoveL Offs(pOrigin,147.63,127.40,0.00),v60,z0,tPen\WObj:=wPaper;
    MoveL Offs(pOrigin,148.52,128.78,0.00),v40,z0,tPen\WObj:=wPaper;
    MoveL Offs(pOrigin,149.86,133.88,0.00),v40,z0,tPen\WObj:=wPaper;
    MoveL Offs(pOrigin,149.86,135.69,0.00),v40,z0,tPen\WObj:=wPaper;
    MoveL Offs(pOrigin,148.91,137.78,0.00),v40,z0,tPen\WObj:=wPaper;
    MoveL Offs(pOrigin,148.16,138.13,0.00),v40,z0,tPen\WObj:=wPaper;
    MoveL Offs(pOrigin,146.78,137.39,0.00),v40,z0,tPen\WObj:=wPaper;
    MoveL Offs(pOrigin,145.58,135.58,0.00),v40,z0,tPen\WObj:=wPaper;
    MoveL Offs(pOrigin,144.98,133.35,0.00),v40,z0,tPen\WObj:=wPaper;
    MoveL Offs(pOrigin,144.98,133.35,0.00),v40,z0,tPen\WObj:=wPaper;
    MoveL Offs(pOrigin,144.66,132.85,0.00),v40,z0,tPen\WObj:=wPaper;
    MoveL Offs(pOrigin,143.91,133.46,0.00),v40,z0,tPen\WObj:=wPaper;
    MoveL Offs(pOrigin,143.91,133.46,0.00),v40,z0,tPen\WObj:=wPaper;
    MoveL Offs(pOrigin,143.81,134.52,0.00),v40,z0,tPen\WObj:=wPaper;
    MoveL Offs(pOrigin,144.12,135.37,0.00),v40,z0,tPen\WObj:=wPaper;
    MoveL Offs(pOrigin,143.81,134.73,0.00),v40,z0,tPen\WObj:=wPaper;
    MoveL Offs(pOrigin,143.17,135.05,0.00),v40,z0,tPen\WObj:=wPaper;
    MoveL Offs(pOrigin,142.96,135.90,0.00),v40,z0,tPen\WObj:=wPaper;
    MoveL Offs(pOrigin,142.96,135.90,0.00),v40,z0,tPen\WObj:=wPaper;
    MoveL Offs(pOrigin,144.02,136.11,0.00),v40,z0,tPen\WObj:=wPaper;
    MoveL Offs(pOrigin,143.91,136.54,0.00),v40,z0,tPen\WObj:=wPaper;
    MoveL Offs(pOrigin,144.02,137.81,0.00),v40,z0,tPen\WObj:=wPaper;
    MoveL Offs(pOrigin,144.02,137.81,0.00),v40,z0,tPen\WObj:=wPaper;
    MoveL Offs(pOrigin,142.53,137.78,0.00),v40,z0,tPen\WObj:=wPaper;
    MoveL Offs(pOrigin,142.74,136.64,0.00),v40,z0,tPen\WObj:=wPaper;
    MoveL Offs(pOrigin,142.74,136.64,0.00),v40,z0,tPen\WObj:=wPaper;
    MoveL Offs(pOrigin,143.91,136.54,0.00),v40,fine,tPen\WObj:=wPaper;
    MoveL Offs(pOrigin,143.91,136.54,6.00),v60,z5,tPen\WObj:=wPaper;
    MoveL Offs(pOrigin,144.44,137.92,6.00),vTravel,z5,tPen\WObj:=wPaper;
    MoveL Offs(pOrigin,144.44,137.92,0.00),v60,z0,tPen\WObj:=wPaper;
    MoveL Offs(pOrigin,144.66,138.63,0.00),v40,z0,tPen\WObj:=wPaper;
    MoveL Offs(pOrigin,146.57,139.51,0.00),v40,z0,tPen\WObj:=wPaper;
    MoveL Offs(pOrigin,147.10,140.36,0.00),v40,z0,tPen\WObj:=wPaper;
    MoveL Offs(pOrigin,147.31,140.36,0.00),v40,z0,tPen\WObj:=wPaper;
    MoveL Offs(pOrigin,147.74,140.04,0.00),v40,z0,tPen\WObj:=wPaper;
    MoveL Offs(pOrigin,148.91,140.15,0.00),v40,z0,tPen\WObj:=wPaper;
    MoveL Offs(pOrigin,148.91,140.15,0.00),v40,z0,tPen\WObj:=wPaper;
    MoveL Offs(pOrigin,149.33,140.47,0.00),v40,z0,tPen\WObj:=wPaper;
    MoveL Offs(pOrigin,149.01,141.96,0.00),v40,z0,tPen\WObj:=wPaper;
    MoveL Offs(pOrigin,148.80,141.96,0.00),v40,z0,tPen\WObj:=wPaper;
    MoveL Offs(pOrigin,149.12,143.34,0.00),v40,z0,tPen\WObj:=wPaper;
    MoveL Offs(pOrigin,148.27,143.23,0.00),v40,z0,tPen\WObj:=wPaper;
    MoveL Offs(pOrigin,147.21,141.53,0.00),v40,z0,tPen\WObj:=wPaper;
    MoveL Offs(pOrigin,147.21,141.53,0.00),v40,z0,tPen\WObj:=wPaper;
    MoveL Offs(pOrigin,144.66,141.21,0.00),v40,z0,tPen\WObj:=wPaper;
    MoveL Offs(pOrigin,144.66,141.21,0.00),v40,z0,tPen\WObj:=wPaper;
    MoveL Offs(pOrigin,145.40,140.57,0.00),v40,z0,tPen\WObj:=wPaper;
    MoveL Offs(pOrigin,145.40,140.57,0.00),v40,z0,tPen\WObj:=wPaper;
    MoveL Offs(pOrigin,147.21,140.43,0.00),v40,z0,tPen\WObj:=wPaper;
    MoveL Offs(pOrigin,147.42,141.11,0.00),v40,z0,tPen\WObj:=wPaper;
    MoveL Offs(pOrigin,148.27,141.00,0.00),v40,z0,tPen\WObj:=wPaper;
    MoveL Offs(pOrigin,148.80,141.96,0.00),v40,z0,tPen\WObj:=wPaper;
    MoveL Offs(pOrigin,148.80,141.96,0.00),v40,z0,tPen\WObj:=wPaper;
    MoveL Offs(pOrigin,147.84,142.06,0.00),v40,z0,tPen\WObj:=wPaper;
    MoveL Offs(pOrigin,148.27,141.00,0.00),v40,z0,tPen\WObj:=wPaper;
    MoveL Offs(pOrigin,148.91,140.36,0.00),v40,z0,tPen\WObj:=wPaper;
    MoveL Offs(pOrigin,149.33,140.26,0.00),v40,z0,tPen\WObj:=wPaper;
    MoveL Offs(pOrigin,150.75,137.49,0.00),v40,z0,tPen\WObj:=wPaper;
    MoveL Offs(pOrigin,151.35,134.52,0.00),v40,z0,tPen\WObj:=wPaper;
    MoveL Offs(pOrigin,149.33,125.38,0.00),v40,z0,tPen\WObj:=wPaper;
    MoveL Offs(pOrigin,149.33,125.38,0.00),v40,z0,tPen\WObj:=wPaper;
    MoveL Offs(pOrigin,163.99,125.17,0.00),v40,z0,tPen\WObj:=wPaper;
    MoveL Offs(pOrigin,179.08,123.79,0.00),v40,z0,tPen\WObj:=wPaper;
    MoveL Offs(pOrigin,183.23,123.04,0.00),v40,z0,tPen\WObj:=wPaper;
    MoveL Offs(pOrigin,186.31,122.02,0.00),v40,z0,tPen\WObj:=wPaper;
    MoveL Offs(pOrigin,187.90,120.99,0.00),v40,z0,tPen\WObj:=wPaper;
    MoveL Offs(pOrigin,188.64,119.75,0.00),v40,fine,tPen\WObj:=wPaper;
    MoveL Offs(pOrigin,188.64,119.75,6.00),v60,z5,tPen\WObj:=wPaper;
    MoveL Offs(pOrigin,179.19,122.30,6.00),vTravel,z5,tPen\WObj:=wPaper;
    MoveL Offs(pOrigin,179.19,122.30,0.00),v60,z0,tPen\WObj:=wPaper;
    MoveL Offs(pOrigin,181.52,122.09,0.00),v40,z0,tPen\WObj:=wPaper;
    MoveL Offs(pOrigin,183.65,121.49,0.00),v40,z0,tPen\WObj:=wPaper;
    MoveL Offs(pOrigin,185.46,120.56,0.00),v40,z0,tPen\WObj:=wPaper;
    MoveL Offs(pOrigin,186.62,119.43,0.00),v40,z0,tPen\WObj:=wPaper;
    MoveL Offs(pOrigin,187.51,117.84,0.00),v40,z0,tPen\WObj:=wPaper;
    MoveL Offs(pOrigin,188.22,115.29,0.00),v40,z0,tPen\WObj:=wPaper;
    MoveL Offs(pOrigin,188.54,112.42,0.00),v40,z0,tPen\WObj:=wPaper;
    MoveL Offs(pOrigin,188.32,109.02,0.00),v40,z0,tPen\WObj:=wPaper;
    MoveL Offs(pOrigin,188.32,109.02,0.00),v40,z0,tPen\WObj:=wPaper;
    MoveL Offs(pOrigin,188.11,105.62,0.00),v40,z0,tPen\WObj:=wPaper;
    MoveL Offs(pOrigin,186.52,97.44,0.00),v40,z0,tPen\WObj:=wPaper;
    MoveL Offs(pOrigin,186.52,97.44,0.00),v40,z0,tPen\WObj:=wPaper;
    MoveL Offs(pOrigin,185.35,97.44,0.00),v40,z0,tPen\WObj:=wPaper;
    MoveL Offs(pOrigin,185.35,97.44,0.00),v40,z0,tPen\WObj:=wPaper;
    MoveL Offs(pOrigin,183.51,94.14,0.00),v40,z0,tPen\WObj:=wPaper;
    MoveL Offs(pOrigin,181.42,87.98,0.00),v40,z0,tPen\WObj:=wPaper;
    MoveL Offs(pOrigin,177.81,74.38,0.00),v40,z0,tPen\WObj:=wPaper;
    MoveL Offs(pOrigin,176.32,66.84,0.00),v40,z0,tPen\WObj:=wPaper;
    MoveL Offs(pOrigin,176.32,66.84,0.00),v40,z0,tPen\WObj:=wPaper;
    MoveL Offs(pOrigin,176.96,67.26,0.00),v40,z0,tPen\WObj:=wPaper;
    MoveL Offs(pOrigin,178.34,69.39,0.00),v40,z0,tPen\WObj:=wPaper;
    MoveL Offs(pOrigin,181.42,73.00,0.00),v40,z0,tPen\WObj:=wPaper;
    MoveL Offs(pOrigin,183.97,75.34,0.00),v40,z0,tPen\WObj:=wPaper;
    MoveL Offs(pOrigin,187.48,77.78,0.00),v40,fine,tPen\WObj:=wPaper;
    MoveL Offs(pOrigin,187.48,77.78,6.00),v60,z5,tPen\WObj:=wPaper;
    MoveL Offs(pOrigin,188.32,74.49,6.00),vTravel,z5,tPen\WObj:=wPaper;
    MoveL Offs(pOrigin,188.32,74.49,0.00),v60,z0,tPen\WObj:=wPaper;
  ENDPROC

  PROC DrawPart6()
    MoveL Offs(pOrigin,185.14,73.25,0.00),v40,z0,tPen\WObj:=wPaper;
    MoveL Offs(pOrigin,183.23,72.04,0.00),v40,z0,tPen\WObj:=wPaper;
    MoveL Offs(pOrigin,178.98,67.90,0.00),v40,z0,tPen\WObj:=wPaper;
    MoveL Offs(pOrigin,176.64,64.29,0.00),v40,z0,tPen\WObj:=wPaper;
    MoveL Offs(pOrigin,175.93,63.76,0.00),v40,z0,tPen\WObj:=wPaper;
    MoveL Offs(pOrigin,174.62,58.66,0.00),v40,z0,tPen\WObj:=wPaper;
    MoveL Offs(pOrigin,174.51,56.96,0.00),v40,z0,tPen\WObj:=wPaper;
    MoveL Offs(pOrigin,174.51,56.96,0.00),v40,z0,tPen\WObj:=wPaper;
    MoveL Offs(pOrigin,174.09,55.36,0.00),v40,z0,tPen\WObj:=wPaper;
    MoveL Offs(pOrigin,174.09,55.36,0.00),v40,z0,tPen\WObj:=wPaper;
    MoveL Offs(pOrigin,174.30,53.24,0.00),v40,z0,tPen\WObj:=wPaper;
    MoveL Offs(pOrigin,178.76,56.74,0.00),v40,z0,tPen\WObj:=wPaper;
    MoveL Offs(pOrigin,183.23,59.44,0.00),v40,z0,tPen\WObj:=wPaper;
    MoveL Offs(pOrigin,189.81,62.73,0.00),v40,z0,tPen\WObj:=wPaper;
    MoveL Offs(pOrigin,193.64,64.07,0.00),v40,fine,tPen\WObj:=wPaper;
    MoveL Offs(pOrigin,193.64,64.07,6.00),v60,z5,tPen\WObj:=wPaper;
    MoveL Offs(pOrigin,195.44,66.41,6.00),vTravel,z5,tPen\WObj:=wPaper;
    MoveL Offs(pOrigin,195.44,66.41,0.00),v60,z0,tPen\WObj:=wPaper;
    MoveL Offs(pOrigin,194.70,72.36,0.00),v40,z0,tPen\WObj:=wPaper;
    MoveL Offs(pOrigin,192.89,74.70,0.00),v40,z0,tPen\WObj:=wPaper;
    MoveL Offs(pOrigin,192.89,74.70,0.00),v40,z0,tPen\WObj:=wPaper;
    MoveL Offs(pOrigin,193.11,77.25,0.00),v40,z0,tPen\WObj:=wPaper;
    MoveL Offs(pOrigin,189.88,85.22,0.00),v40,z0,tPen\WObj:=wPaper;
    MoveL Offs(pOrigin,190.45,88.09,0.00),v40,z0,tPen\WObj:=wPaper;
    MoveL Offs(pOrigin,189.39,91.17,0.00),v40,z0,tPen\WObj:=wPaper;
    MoveL Offs(pOrigin,188.75,94.68,0.00),v40,z0,tPen\WObj:=wPaper;
    MoveL Offs(pOrigin,189.28,95.31,0.00),v40,z0,tPen\WObj:=wPaper;
    MoveL Offs(pOrigin,190.56,106.79,0.00),v40,z0,tPen\WObj:=wPaper;
    MoveL Offs(pOrigin,190.34,113.80,0.00),v40,z0,tPen\WObj:=wPaper;
    MoveL Offs(pOrigin,189.92,116.35,0.00),v40,z0,tPen\WObj:=wPaper;
    MoveL Offs(pOrigin,188.68,119.43,0.00),v40,z0,tPen\WObj:=wPaper;
    MoveL Offs(pOrigin,189.07,119.96,0.00),v40,z0,tPen\WObj:=wPaper;
    MoveL Offs(pOrigin,191.02,117.20,0.00),v40,z0,tPen\WObj:=wPaper;
    MoveL Offs(pOrigin,192.47,111.78,0.00),v40,z0,tPen\WObj:=wPaper;
    MoveL Offs(pOrigin,196.72,66.41,0.00),v40,z0,tPen\WObj:=wPaper;
    MoveL Offs(pOrigin,196.72,66.41,0.00),v40,z0,tPen\WObj:=wPaper;
    MoveL Offs(pOrigin,197.85,65.67,0.00),v40,z0,tPen\WObj:=wPaper;
    MoveL Offs(pOrigin,198.17,61.10,0.00),v40,z0,tPen\WObj:=wPaper;
    MoveL Offs(pOrigin,199.84,58.44,0.00),v40,z0,tPen\WObj:=wPaper;
    MoveL Offs(pOrigin,200.51,55.58,0.00),v40,z0,tPen\WObj:=wPaper;
    MoveL Offs(pOrigin,203.24,51.33,0.00),v40,z0,tPen\WObj:=wPaper;
    MoveL Offs(pOrigin,205.01,44.74,0.00),v40,z0,tPen\WObj:=wPaper;
    MoveL Offs(pOrigin,207.13,39.21,0.00),v40,z0,tPen\WObj:=wPaper;
    MoveL Offs(pOrigin,207.56,37.41,0.00),v40,z0,tPen\WObj:=wPaper;
    MoveL Offs(pOrigin,207.34,34.86,0.00),v40,z0,tPen\WObj:=wPaper;
    MoveL Offs(pOrigin,207.88,31.35,0.00),v40,z0,tPen\WObj:=wPaper;
    MoveL Offs(pOrigin,207.34,27.63,0.00),v40,z0,tPen\WObj:=wPaper;
    MoveL Offs(pOrigin,205.54,24.12,0.00),v40,z0,tPen\WObj:=wPaper;
    MoveL Offs(pOrigin,203.73,22.71,0.00),v40,z0,tPen\WObj:=wPaper;
    MoveL Offs(pOrigin,201.93,21.86,0.00),v40,z0,tPen\WObj:=wPaper;
    MoveL Offs(pOrigin,198.63,20.83,0.00),v40,z0,tPen\WObj:=wPaper;
    MoveL Offs(pOrigin,192.89,19.66,0.00),v40,z0,tPen\WObj:=wPaper;
    MoveL Offs(pOrigin,183.12,18.39,0.00),v40,z0,tPen\WObj:=wPaper;
    MoveL Offs(pOrigin,182.80,18.60,0.00),v40,z0,tPen\WObj:=wPaper;
    MoveL Offs(pOrigin,182.80,18.60,0.00),v40,z0,tPen\WObj:=wPaper;
    MoveL Offs(pOrigin,183.33,19.27,0.00),v40,z0,tPen\WObj:=wPaper;
    MoveL Offs(pOrigin,192.04,21.79,0.00),v40,fine,tPen\WObj:=wPaper;
    MoveL Offs(pOrigin,192.04,21.79,6.00),v60,z5,tPen\WObj:=wPaper;
    MoveL Offs(pOrigin,192.15,25.72,6.00),vTravel,z5,tPen\WObj:=wPaper;
    MoveL Offs(pOrigin,192.15,25.72,0.00),v60,z0,tPen\WObj:=wPaper;
    MoveL Offs(pOrigin,188.86,28.91,0.00),v40,z0,tPen\WObj:=wPaper;
    MoveL Offs(pOrigin,188.64,29.01,0.00),v40,z0,tPen\WObj:=wPaper;
    MoveL Offs(pOrigin,185.77,31.46,0.00),v40,fine,tPen\WObj:=wPaper;
    MoveL Offs(pOrigin,185.77,31.46,6.00),v60,z5,tPen\WObj:=wPaper;
    MoveL Offs(pOrigin,188.96,31.35,6.00),vTravel,z5,tPen\WObj:=wPaper;
    MoveL Offs(pOrigin,188.96,31.35,0.00),v60,z0,tPen\WObj:=wPaper;
    MoveL Offs(pOrigin,185.46,34.04,0.00),v40,z0,tPen\WObj:=wPaper;
    MoveL Offs(pOrigin,180.78,36.49,0.00),v40,z0,tPen\WObj:=wPaper;
    MoveL Offs(pOrigin,174.83,38.36,0.00),v40,z0,tPen\WObj:=wPaper;
    MoveL Offs(pOrigin,170.90,38.89,0.00),v40,fine,tPen\WObj:=wPaper;
    MoveL Offs(pOrigin,170.90,38.89,6.00),v60,z5,tPen\WObj:=wPaper;
    MoveL Offs(pOrigin,168.99,39.85,6.00),vTravel,z5,tPen\WObj:=wPaper;
    MoveL Offs(pOrigin,168.99,39.85,0.00),v60,z0,tPen\WObj:=wPaper;
    MoveL Offs(pOrigin,159.64,38.04,0.00),v40,z0,tPen\WObj:=wPaper;
    MoveL Offs(pOrigin,156.98,37.02,0.00),v40,z0,tPen\WObj:=wPaper;
    MoveL Offs(pOrigin,156.56,36.34,0.00),v40,z0,tPen\WObj:=wPaper;
    MoveL Offs(pOrigin,156.56,36.34,0.00),v40,z0,tPen\WObj:=wPaper;
    MoveL Offs(pOrigin,160.49,36.56,0.00),v40,z0,tPen\WObj:=wPaper;
    MoveL Offs(pOrigin,164.21,35.32,0.00),v40,z0,tPen\WObj:=wPaper;
    MoveL Offs(pOrigin,167.71,33.05,0.00),v40,z0,tPen\WObj:=wPaper;
    MoveL Offs(pOrigin,171.22,29.33,0.00),v40,z0,tPen\WObj:=wPaper;
    MoveL Offs(pOrigin,173.91,24.98,0.00),v40,z0,tPen\WObj:=wPaper;
    MoveL Offs(pOrigin,175.15,21.36,0.00),v40,z0,tPen\WObj:=wPaper;
    MoveL Offs(pOrigin,174.65,18.28,0.00),v40,z0,tPen\WObj:=wPaper;
    MoveL Offs(pOrigin,173.56,16.58,0.00),v40,z0,tPen\WObj:=wPaper;
    MoveL Offs(pOrigin,172.28,15.62,0.00),v40,z0,tPen\WObj:=wPaper;
    MoveL Offs(pOrigin,171.96,14.99,0.00),v40,fine,tPen\WObj:=wPaper;
    MoveL Offs(pOrigin,171.96,14.99,6.00),v60,z5,tPen\WObj:=wPaper;
    MoveL Offs(pOrigin,171.22,16.65,6.00),vTravel,z5,tPen\WObj:=wPaper;
    MoveL Offs(pOrigin,171.22,16.65,0.00),v60,z0,tPen\WObj:=wPaper;
    MoveL Offs(pOrigin,171.71,17.01,0.00),v40,z0,tPen\WObj:=wPaper;
    MoveL Offs(pOrigin,171.61,17.54,0.00),v40,z0,tPen\WObj:=wPaper;
    MoveL Offs(pOrigin,170.26,17.25,0.00),v40,z0,tPen\WObj:=wPaper;
    MoveL Offs(pOrigin,169.84,16.58,0.00),v40,z0,tPen\WObj:=wPaper;
    MoveL Offs(pOrigin,171.22,16.65,0.00),v40,z0,tPen\WObj:=wPaper;
    MoveL Offs(pOrigin,171.75,17.54,0.00),v40,z0,tPen\WObj:=wPaper;
    MoveL Offs(pOrigin,173.27,19.34,0.00),v40,z0,tPen\WObj:=wPaper;
    MoveL Offs(pOrigin,174.41,22.85,0.00),v40,fine,tPen\WObj:=wPaper;
    MoveL Offs(pOrigin,174.41,22.85,6.00),v60,z5,tPen\WObj:=wPaper;
    MoveL Offs(pOrigin,177.27,22.21,6.00),vTravel,z5,tPen\WObj:=wPaper;
    MoveL Offs(pOrigin,177.27,22.21,0.00),v60,z0,tPen\WObj:=wPaper;
    MoveL Offs(pOrigin,176.43,19.24,0.00),v40,fine,tPen\WObj:=wPaper;
    MoveL Offs(pOrigin,176.43,19.24,6.00),v60,z5,tPen\WObj:=wPaper;
    MoveL Offs(pOrigin,170.94,19.66,6.00),vTravel,z5,tPen\WObj:=wPaper;
    MoveL Offs(pOrigin,170.94,19.66,0.00),v60,z0,tPen\WObj:=wPaper;
    MoveL Offs(pOrigin,171.22,21.04,0.00),v40,z0,tPen\WObj:=wPaper;
    MoveL Offs(pOrigin,170.79,21.75,0.00),v40,z0,tPen\WObj:=wPaper;
    MoveL Offs(pOrigin,169.73,21.82,0.00),v40,z0,tPen\WObj:=wPaper;
    MoveL Offs(pOrigin,168.85,20.94,0.00),v40,z0,tPen\WObj:=wPaper;
    MoveL Offs(pOrigin,168.56,19.88,0.00),v40,z0,tPen\WObj:=wPaper;
    MoveL Offs(pOrigin,169.31,18.99,0.00),v40,z0,tPen\WObj:=wPaper;
    MoveL Offs(pOrigin,170.26,19.06,0.00),v40,z0,tPen\WObj:=wPaper;
    MoveL Offs(pOrigin,170.94,19.66,0.00),v40,fine,tPen\WObj:=wPaper;
    MoveL Offs(pOrigin,170.94,19.66,6.00),v60,z5,tPen\WObj:=wPaper;
    MoveL Offs(pOrigin,169.09,20.19,6.00),vTravel,z5,tPen\WObj:=wPaper;
    MoveL Offs(pOrigin,169.09,20.19,0.00),v60,z0,tPen\WObj:=wPaper;
    MoveL Offs(pOrigin,169.62,21.26,0.00),v40,fine,tPen\WObj:=wPaper;
    MoveL Offs(pOrigin,169.62,21.26,6.00),v60,z5,tPen\WObj:=wPaper;
    MoveL Offs(pOrigin,169.73,16.79,6.00),vTravel,z5,tPen\WObj:=wPaper;
    MoveL Offs(pOrigin,169.73,16.79,0.00),v60,z0,tPen\WObj:=wPaper;
  ENDPROC

  PROC DrawPart7()
    MoveL Offs(pOrigin,167.93,16.58,0.00),v40,z0,tPen\WObj:=wPaper;
    MoveL Offs(pOrigin,167.50,16.26,0.00),v40,z0,tPen\WObj:=wPaper;
    MoveL Offs(pOrigin,167.50,16.26,0.00),v40,z0,tPen\WObj:=wPaper;
    MoveL Offs(pOrigin,167.93,15.70,0.00),v40,z0,tPen\WObj:=wPaper;
    MoveL Offs(pOrigin,169.62,15.09,0.00),v40,z0,tPen\WObj:=wPaper;
    MoveL Offs(pOrigin,172.71,14.88,0.00),v40,z0,tPen\WObj:=wPaper;
    MoveL Offs(pOrigin,182.80,18.60,0.00),v40,fine,tPen\WObj:=wPaper;
    MoveL Offs(pOrigin,182.80,18.60,6.00),v60,z5,tPen\WObj:=wPaper;
    MoveL Offs(pOrigin,191.51,28.91,6.00),vTravel,z5,tPen\WObj:=wPaper;
    MoveL Offs(pOrigin,191.51,28.91,0.00),v60,z0,tPen\WObj:=wPaper;
    MoveL Offs(pOrigin,189.18,31.24,0.00),v40,fine,tPen\WObj:=wPaper;
    MoveL Offs(pOrigin,189.18,31.24,6.00),v60,z5,tPen\WObj:=wPaper;
    MoveL Offs(pOrigin,194.81,36.03,6.00),vTravel,z5,tPen\WObj:=wPaper;
    MoveL Offs(pOrigin,194.81,36.03,0.00),v60,z0,tPen\WObj:=wPaper;
    MoveL Offs(pOrigin,194.49,36.34,0.00),v40,z0,tPen\WObj:=wPaper;
    MoveL Offs(pOrigin,194.81,36.03,0.00),v40,z0,tPen\WObj:=wPaper;
    MoveL Offs(pOrigin,195.44,35.49,0.00),v40,z0,tPen\WObj:=wPaper;
    MoveL Offs(pOrigin,191.94,38.29,0.00),v40,z0,tPen\WObj:=wPaper;
    MoveL Offs(pOrigin,188.96,39.78,0.00),v40,z0,tPen\WObj:=wPaper;
    MoveL Offs(pOrigin,186.41,40.49,0.00),v40,z0,tPen\WObj:=wPaper;
    MoveL Offs(pOrigin,180.89,41.12,0.00),v40,fine,tPen\WObj:=wPaper;
    MoveL Offs(pOrigin,180.89,41.12,6.00),v60,z5,tPen\WObj:=wPaper;
    MoveL Offs(pOrigin,183.54,42.29,6.00),vTravel,z5,tPen\WObj:=wPaper;
    MoveL Offs(pOrigin,183.54,42.29,0.00),v60,z0,tPen\WObj:=wPaper;
    MoveL Offs(pOrigin,188.11,42.72,0.00),v40,z0,tPen\WObj:=wPaper;
    MoveL Offs(pOrigin,192.89,41.76,0.00),v40,fine,tPen\WObj:=wPaper;
    MoveL Offs(pOrigin,192.89,41.76,6.00),v60,z5,tPen\WObj:=wPaper;
    MoveL Offs(pOrigin,190.98,45.06,6.00),vTravel,z5,tPen\WObj:=wPaper;
    MoveL Offs(pOrigin,190.98,45.06,0.00),v60,z0,tPen\WObj:=wPaper;
    MoveL Offs(pOrigin,197.25,42.97,0.00),v40,z0,tPen\WObj:=wPaper;
    MoveL Offs(pOrigin,202.99,39.53,0.00),v40,z0,tPen\WObj:=wPaper;
    MoveL Offs(pOrigin,203.20,39.42,0.00),v40,z0,tPen\WObj:=wPaper;
    MoveL Offs(pOrigin,207.34,35.49,0.00),v40,fine,tPen\WObj:=wPaper;
    MoveL Offs(pOrigin,207.34,35.49,6.00),v60,z5,tPen\WObj:=wPaper;
    MoveL Offs(pOrigin,203.62,36.13,6.00),vTravel,z5,tPen\WObj:=wPaper;
    MoveL Offs(pOrigin,203.62,36.13,0.00),v60,z0,tPen\WObj:=wPaper;
    MoveL Offs(pOrigin,202.35,37.94,0.00),v40,z0,tPen\WObj:=wPaper;
    MoveL Offs(pOrigin,201.50,38.15,0.00),v40,z0,tPen\WObj:=wPaper;
    MoveL Offs(pOrigin,203.34,35.07,0.00),v40,z0,tPen\WObj:=wPaper;
    MoveL Offs(pOrigin,204.79,30.82,0.00),v40,z0,tPen\WObj:=wPaper;
    MoveL Offs(pOrigin,204.90,26.78,0.00),v40,z0,tPen\WObj:=wPaper;
    MoveL Offs(pOrigin,204.05,23.17,0.00),v40,fine,tPen\WObj:=wPaper;
    MoveL Offs(pOrigin,204.05,23.17,6.00),v60,z5,tPen\WObj:=wPaper;
    MoveL Offs(pOrigin,201.18,24.34,6.00),vTravel,z5,tPen\WObj:=wPaper;
    MoveL Offs(pOrigin,201.18,24.34,0.00),v60,z0,tPen\WObj:=wPaper;
    MoveL Offs(pOrigin,200.65,27.42,0.00),v40,z0,tPen\WObj:=wPaper;
    MoveL Offs(pOrigin,199.73,29.76,0.00),v40,z0,tPen\WObj:=wPaper;
    MoveL Offs(pOrigin,197.99,32.62,0.00),v40,z0,tPen\WObj:=wPaper;
    MoveL Offs(pOrigin,195.66,35.39,0.00),v40,fine,tPen\WObj:=wPaper;
    MoveL Offs(pOrigin,195.66,35.39,6.00),v60,z5,tPen\WObj:=wPaper;
    MoveL Offs(pOrigin,205.01,39.64,6.00),vTravel,z5,tPen\WObj:=wPaper;
    MoveL Offs(pOrigin,205.01,39.64,0.00),v60,z0,tPen\WObj:=wPaper;
    MoveL Offs(pOrigin,204.69,39.96,0.00),v40,z0,tPen\WObj:=wPaper;
    MoveL Offs(pOrigin,205.01,39.64,0.00),v40,z0,tPen\WObj:=wPaper;
    MoveL Offs(pOrigin,205.43,39.11,0.00),v40,z0,tPen\WObj:=wPaper;
    MoveL Offs(pOrigin,203.09,41.66,0.00),v40,z0,tPen\WObj:=wPaper;
    MoveL Offs(pOrigin,200.23,43.71,0.00),v40,z0,tPen\WObj:=wPaper;
    MoveL Offs(pOrigin,197.25,44.95,0.00),v40,z0,tPen\WObj:=wPaper;
    MoveL Offs(pOrigin,194.17,45.59,0.00),v40,z0,tPen\WObj:=wPaper;
    MoveL Offs(pOrigin,191.73,45.59,0.00),v40,z0,tPen\WObj:=wPaper;
    MoveL Offs(pOrigin,190.77,45.06,0.00),v40,z0,tPen\WObj:=wPaper;
    MoveL Offs(pOrigin,187.58,44.74,0.00),v40,z0,tPen\WObj:=wPaper;
    MoveL Offs(pOrigin,183.65,43.18,0.00),v40,z0,tPen\WObj:=wPaper;
    MoveL Offs(pOrigin,181.10,41.66,0.00),v40,z0,tPen\WObj:=wPaper;
    MoveL Offs(pOrigin,180.78,41.16,0.00),v40,z0,tPen\WObj:=wPaper;
    MoveL Offs(pOrigin,176.85,40.84,0.00),v40,z0,tPen\WObj:=wPaper;
    MoveL Offs(pOrigin,176.32,43.36,0.00),v40,z0,tPen\WObj:=wPaper;
    MoveL Offs(pOrigin,176.11,47.50,0.00),v40,z0,tPen\WObj:=wPaper;
    MoveL Offs(pOrigin,177.03,50.37,0.00),v40,z0,tPen\WObj:=wPaper;
    MoveL Offs(pOrigin,178.12,52.39,0.00),v40,fine,tPen\WObj:=wPaper;
    MoveL Offs(pOrigin,178.12,52.39,6.00),v60,z5,tPen\WObj:=wPaper;
    MoveL Offs(pOrigin,179.82,51.01,6.00),vTravel,z5,tPen\WObj:=wPaper;
    MoveL Offs(pOrigin,179.82,51.01,0.00),v60,z0,tPen\WObj:=wPaper;
    MoveL Offs(pOrigin,180.78,52.60,0.00),v40,z0,tPen\WObj:=wPaper;
    MoveL Offs(pOrigin,182.80,54.02,0.00),v40,z0,tPen\WObj:=wPaper;
    MoveL Offs(pOrigin,185.56,54.83,0.00),v40,z0,tPen\WObj:=wPaper;
    MoveL Offs(pOrigin,188.96,54.94,0.00),v40,z0,tPen\WObj:=wPaper;
    MoveL Offs(pOrigin,193.32,54.19,0.00),v40,z0,tPen\WObj:=wPaper;
    MoveL Offs(pOrigin,197.14,52.85,0.00),v40,z0,tPen\WObj:=wPaper;
    MoveL Offs(pOrigin,200.23,51.11,0.00),v40,z0,tPen\WObj:=wPaper;
    MoveL Offs(pOrigin,201.93,49.62,0.00),v40,fine,tPen\WObj:=wPaper;
    MoveL Offs(pOrigin,201.93,49.62,6.00),v60,z5,tPen\WObj:=wPaper;
    MoveL Offs(pOrigin,198.21,47.08,6.00),vTravel,z5,tPen\WObj:=wPaper;
    MoveL Offs(pOrigin,198.21,47.08,0.00),v60,z0,tPen\WObj:=wPaper;
    MoveL Offs(pOrigin,193.85,47.39,0.00),v40,z0,tPen\WObj:=wPaper;
    MoveL Offs(pOrigin,189.49,46.22,0.00),v40,fine,tPen\WObj:=wPaper;
    MoveL Offs(pOrigin,189.49,46.22,6.00),v60,z5,tPen\WObj:=wPaper;
    MoveL Offs(pOrigin,186.62,51.01,6.00),vTravel,z5,tPen\WObj:=wPaper;
    MoveL Offs(pOrigin,186.62,51.01,0.00),v60,z0,tPen\WObj:=wPaper;
    MoveL Offs(pOrigin,184.71,50.51,0.00),v40,z0,tPen\WObj:=wPaper;
    MoveL Offs(pOrigin,182.38,49.20,0.00),v40,z0,tPen\WObj:=wPaper;
    MoveL Offs(pOrigin,180.04,47.08,0.00),v40,z0,tPen\WObj:=wPaper;
    MoveL Offs(pOrigin,178.76,45.27,0.00),v40,fine,tPen\WObj:=wPaper;
    MoveL Offs(pOrigin,178.76,45.27,6.00),v60,z5,tPen\WObj:=wPaper;
    MoveL Offs(pOrigin,180.04,46.97,6.00),vTravel,z5,tPen\WObj:=wPaper;
    MoveL Offs(pOrigin,180.04,46.97,0.00),v60,z0,tPen\WObj:=wPaper;
    MoveL Offs(pOrigin,180.57,47.50,0.00),v40,z0,tPen\WObj:=wPaper;
    MoveL Offs(pOrigin,180.04,46.97,0.00),v40,fine,tPen\WObj:=wPaper;
    MoveL Offs(pOrigin,180.04,46.97,6.00),v60,z5,tPen\WObj:=wPaper;
    MoveL Offs(pOrigin,183.54,47.82,6.00),vTravel,z5,tPen\WObj:=wPaper;
    MoveL Offs(pOrigin,183.54,47.82,0.00),v60,z0,tPen\WObj:=wPaper;
    MoveL Offs(pOrigin,179.82,44.63,0.00),v40,z0,tPen\WObj:=wPaper;
    MoveL Offs(pOrigin,177.81,41.66,0.00),v40,fine,tPen\WObj:=wPaper;
    MoveL Offs(pOrigin,177.81,41.66,6.00),v60,z5,tPen\WObj:=wPaper;
    MoveL Offs(pOrigin,176.64,40.91,6.00),vTravel,z5,tPen\WObj:=wPaper;
    MoveL Offs(pOrigin,176.64,40.91,0.00),v60,z0,tPen\WObj:=wPaper;
    MoveL Offs(pOrigin,173.88,40.59,0.00),v40,z0,tPen\WObj:=wPaper;
    MoveL Offs(pOrigin,173.88,40.59,0.00),v40,z0,tPen\WObj:=wPaper;
    MoveL Offs(pOrigin,174.94,48.67,0.00),v40,z0,tPen\WObj:=wPaper;
    MoveL Offs(pOrigin,174.94,48.67,0.00),v40,z0,tPen\WObj:=wPaper;
    MoveL Offs(pOrigin,173.88,52.07,0.00),v40,z0,tPen\WObj:=wPaper;
    MoveL Offs(pOrigin,173.88,52.07,0.00),v40,z0,tPen\WObj:=wPaper;
    MoveL Offs(pOrigin,174.09,53.24,0.00),v40,z0,tPen\WObj:=wPaper;
    MoveL Offs(pOrigin,173.88,52.07,0.00),v40,z0,tPen\WObj:=wPaper;
    MoveL Offs(pOrigin,173.31,51.75,0.00),v40,z0,tPen\WObj:=wPaper;
    MoveL Offs(pOrigin,172.00,47.50,0.00),v40,z0,tPen\WObj:=wPaper;
    MoveL Offs(pOrigin,168.99,39.85,0.00),v40,z0,tPen\WObj:=wPaper;
    MoveL Offs(pOrigin,168.99,39.85,0.00),v40,z0,tPen\WObj:=wPaper;
    MoveL Offs(pOrigin,173.88,40.59,0.00),v40,fine,tPen\WObj:=wPaper;
    MoveL Offs(pOrigin,173.88,40.59,6.00),v60,z5,tPen\WObj:=wPaper;
  ENDPROC

  PROC DrawPart8()
    MoveL Offs(pOrigin,167.61,41.12,6.00),vTravel,z5,tPen\WObj:=wPaper;
    MoveL Offs(pOrigin,167.61,41.12,0.00),v60,z0,tPen\WObj:=wPaper;
    MoveL Offs(pOrigin,170.72,48.03,0.00),v40,z0,tPen\WObj:=wPaper;
    MoveL Offs(pOrigin,173.20,54.72,0.00),v40,z0,tPen\WObj:=wPaper;
    MoveL Offs(pOrigin,174.09,55.36,0.00),v40,z0,tPen\WObj:=wPaper;
    MoveL Offs(pOrigin,174.41,56.21,0.00),v40,z0,tPen\WObj:=wPaper;
    MoveL Offs(pOrigin,175.47,56.53,0.00),v40,z0,tPen\WObj:=wPaper;
    MoveL Offs(pOrigin,176.85,57.91,0.00),v40,z0,tPen\WObj:=wPaper;
    MoveL Offs(pOrigin,179.61,59.75,0.00),v40,z0,tPen\WObj:=wPaper;
    MoveL Offs(pOrigin,184.18,61.63,0.00),v40,fine,tPen\WObj:=wPaper;
    MoveL Offs(pOrigin,184.18,61.63,6.00),v60,z5,tPen\WObj:=wPaper;
    MoveL Offs(pOrigin,183.54,66.41,6.00),vTravel,z5,tPen\WObj:=wPaper;
    MoveL Offs(pOrigin,183.54,66.41,0.00),v60,z0,tPen\WObj:=wPaper;
    MoveL Offs(pOrigin,181.10,64.82,0.00),v40,z0,tPen\WObj:=wPaper;
    MoveL Offs(pOrigin,178.34,62.16,0.00),v40,z0,tPen\WObj:=wPaper;
    MoveL Offs(pOrigin,175.26,57.49,0.00),v40,z0,tPen\WObj:=wPaper;
    MoveL Offs(pOrigin,174.51,56.96,0.00),v40,fine,tPen\WObj:=wPaper;
    MoveL Offs(pOrigin,174.51,56.96,6.00),v60,z5,tPen\WObj:=wPaper;
    MoveL Offs(pOrigin,176.00,54.41,6.00),vTravel,z5,tPen\WObj:=wPaper;
    MoveL Offs(pOrigin,176.00,54.41,0.00),v60,z0,tPen\WObj:=wPaper;
    MoveL Offs(pOrigin,176.64,55.04,0.00),v40,z0,tPen\WObj:=wPaper;
    MoveL Offs(pOrigin,176.00,54.41,0.00),v40,fine,tPen\WObj:=wPaper;
    MoveL Offs(pOrigin,176.00,54.41,6.00),v60,z5,tPen\WObj:=wPaper;
    MoveL Offs(pOrigin,179.29,55.04,6.00),vTravel,z5,tPen\WObj:=wPaper;
    MoveL Offs(pOrigin,179.29,55.04,0.00),v60,z0,tPen\WObj:=wPaper;
    MoveL Offs(pOrigin,183.12,56.42,0.00),v40,z0,tPen\WObj:=wPaper;
    MoveL Offs(pOrigin,186.41,56.85,0.00),v40,z0,tPen\WObj:=wPaper;
    MoveL Offs(pOrigin,190.77,56.64,0.00),v40,z0,tPen\WObj:=wPaper;
    MoveL Offs(pOrigin,195.66,55.36,0.00),v40,fine,tPen\WObj:=wPaper;
    MoveL Offs(pOrigin,195.66,55.36,6.00),v60,z5,tPen\WObj:=wPaper;
    MoveL Offs(pOrigin,198.31,56.74,6.00),vTravel,z5,tPen\WObj:=wPaper;
    MoveL Offs(pOrigin,198.31,56.74,0.00),v60,z0,tPen\WObj:=wPaper;
    MoveL Offs(pOrigin,195.55,58.16,0.00),v40,z0,tPen\WObj:=wPaper;
    MoveL Offs(pOrigin,191.73,59.08,0.00),v40,fine,tPen\WObj:=wPaper;
    MoveL Offs(pOrigin,191.73,59.08,6.00),v60,z5,tPen\WObj:=wPaper;
    MoveL Offs(pOrigin,189.71,64.82,6.00),vTravel,z5,tPen\WObj:=wPaper;
    MoveL Offs(pOrigin,189.71,64.82,0.00),v60,z0,tPen\WObj:=wPaper;
    MoveL Offs(pOrigin,195.66,66.41,0.00),v40,z0,tPen\WObj:=wPaper;
    MoveL Offs(pOrigin,196.72,66.41,0.00),v40,fine,tPen\WObj:=wPaper;
    MoveL Offs(pOrigin,196.72,66.41,6.00),v60,z5,tPen\WObj:=wPaper;
    MoveL Offs(pOrigin,193.43,71.19,6.00),vTravel,z5,tPen\WObj:=wPaper;
    MoveL Offs(pOrigin,193.43,71.19,0.00),v60,z0,tPen\WObj:=wPaper;
    MoveL Offs(pOrigin,191.19,70.98,0.00),v40,z0,tPen\WObj:=wPaper;
    MoveL Offs(pOrigin,188.22,69.71,0.00),v40,fine,tPen\WObj:=wPaper;
    MoveL Offs(pOrigin,188.22,69.71,6.00),v60,z5,tPen\WObj:=wPaper;
    MoveL Offs(pOrigin,186.52,69.81,6.00),vTravel,z5,tPen\WObj:=wPaper;
    MoveL Offs(pOrigin,186.52,69.81,0.00),v60,z0,tPen\WObj:=wPaper;
    MoveL Offs(pOrigin,192.04,74.38,0.00),v40,z0,tPen\WObj:=wPaper;
    MoveL Offs(pOrigin,192.89,74.70,0.00),v40,fine,tPen\WObj:=wPaper;
    MoveL Offs(pOrigin,192.89,74.70,6.00),v60,z5,tPen\WObj:=wPaper;
    MoveL Offs(pOrigin,182.91,74.28,6.00),vTravel,z5,tPen\WObj:=wPaper;
    MoveL Offs(pOrigin,182.91,74.28,0.00),v60,z0,tPen\WObj:=wPaper;
    MoveL Offs(pOrigin,183.44,74.81,0.00),v40,z0,tPen\WObj:=wPaper;
    MoveL Offs(pOrigin,182.91,74.28,0.00),v40,fine,tPen\WObj:=wPaper;
    MoveL Offs(pOrigin,182.91,74.28,6.00),v60,z5,tPen\WObj:=wPaper;
    MoveL Offs(pOrigin,179.93,73.21,6.00),vTravel,z5,tPen\WObj:=wPaper;
    MoveL Offs(pOrigin,179.93,73.21,0.00),v60,z0,tPen\WObj:=wPaper;
    MoveL Offs(pOrigin,189.28,84.90,0.00),v40,z0,tPen\WObj:=wPaper;
    MoveL Offs(pOrigin,189.81,85.11,0.00),v40,fine,tPen\WObj:=wPaper;
    MoveL Offs(pOrigin,189.81,85.11,6.00),v60,z5,tPen\WObj:=wPaper;
    MoveL Offs(pOrigin,188.01,89.15,6.00),vTravel,z5,tPen\WObj:=wPaper;
    MoveL Offs(pOrigin,188.01,89.15,0.00),v60,z0,tPen\WObj:=wPaper;
    MoveL Offs(pOrigin,181.52,78.10,0.00),v40,fine,tPen\WObj:=wPaper;
    MoveL Offs(pOrigin,181.52,78.10,6.00),v60,z5,tPen\WObj:=wPaper;
    MoveL Offs(pOrigin,180.57,69.81,6.00),vTravel,z5,tPen\WObj:=wPaper;
    MoveL Offs(pOrigin,180.57,69.81,0.00),v60,z0,tPen\WObj:=wPaper;
    MoveL Offs(pOrigin,181.10,70.34,0.00),v40,z0,tPen\WObj:=wPaper;
    MoveL Offs(pOrigin,180.57,69.81,0.00),v40,fine,tPen\WObj:=wPaper;
    MoveL Offs(pOrigin,180.57,69.81,6.00),v60,z5,tPen\WObj:=wPaper;
    MoveL Offs(pOrigin,176.32,66.84,6.00),vTravel,z5,tPen\WObj:=wPaper;
    MoveL Offs(pOrigin,176.32,66.84,0.00),v60,z0,tPen\WObj:=wPaper;
    MoveL Offs(pOrigin,175.79,64.93,0.00),v40,z0,tPen\WObj:=wPaper;
    MoveL Offs(pOrigin,175.89,63.86,0.00),v40,fine,tPen\WObj:=wPaper;
    MoveL Offs(pOrigin,175.89,63.86,6.00),v60,z5,tPen\WObj:=wPaper;
    MoveL Offs(pOrigin,178.44,62.16,6.00),vTravel,z5,tPen\WObj:=wPaper;
    MoveL Offs(pOrigin,178.44,62.16,0.00),v60,z0,tPen\WObj:=wPaper;
    MoveL Offs(pOrigin,178.87,62.59,0.00),v40,z0,tPen\WObj:=wPaper;
    MoveL Offs(pOrigin,178.44,62.16,0.00),v40,fine,tPen\WObj:=wPaper;
    MoveL Offs(pOrigin,178.44,62.16,6.00),v60,z5,tPen\WObj:=wPaper;
    MoveL Offs(pOrigin,170.90,65.56,6.00),vTravel,z5,tPen\WObj:=wPaper;
    MoveL Offs(pOrigin,170.90,65.56,0.00),v60,z0,tPen\WObj:=wPaper;
    MoveL Offs(pOrigin,150.93,60.14,0.00),v40,fine,tPen\WObj:=wPaper;
    MoveL Offs(pOrigin,150.93,60.14,6.00),v60,z5,tPen\WObj:=wPaper;
    MoveL Offs(pOrigin,148.69,60.89,6.00),vTravel,z5,tPen\WObj:=wPaper;
    MoveL Offs(pOrigin,148.69,60.89,0.00),v60,z0,tPen\WObj:=wPaper;
    MoveL Offs(pOrigin,146.99,55.47,0.00),v40,z0,tPen\WObj:=wPaper;
    MoveL Offs(pOrigin,146.99,55.47,0.00),v40,z0,tPen\WObj:=wPaper;
    MoveL Offs(pOrigin,148.38,55.36,0.00),v40,z0,tPen\WObj:=wPaper;
    MoveL Offs(pOrigin,152.94,56.42,0.00),v40,z0,tPen\WObj:=wPaper;
    MoveL Offs(pOrigin,172.18,61.70,0.00),v40,z0,tPen\WObj:=wPaper;
    MoveL Offs(pOrigin,172.60,62.69,0.00),v40,z0,tPen\WObj:=wPaper;
    MoveL Offs(pOrigin,172.35,67.33,0.00),v40,z0,tPen\WObj:=wPaper;
    MoveL Offs(pOrigin,167.29,65.99,0.00),v40,z0,tPen\WObj:=wPaper;
    MoveL Offs(pOrigin,166.97,66.20,0.00),v40,z0,tPen\WObj:=wPaper;
    MoveL Offs(pOrigin,170.05,68.96,0.00),v40,z0,tPen\WObj:=wPaper;
    MoveL Offs(pOrigin,173.77,71.51,0.00),v40,fine,tPen\WObj:=wPaper;
    MoveL Offs(pOrigin,173.77,71.51,6.00),v60,z5,tPen\WObj:=wPaper;
    MoveL Offs(pOrigin,166.97,65.99,6.00),vTravel,z5,tPen\WObj:=wPaper;
    MoveL Offs(pOrigin,166.97,65.99,0.00),v60,z0,tPen\WObj:=wPaper;
    MoveL Offs(pOrigin,148.80,60.92,0.00),v40,z0,tPen\WObj:=wPaper;
    MoveL Offs(pOrigin,149.01,62.38,0.00),v40,z0,tPen\WObj:=wPaper;
    MoveL Offs(pOrigin,158.89,93.51,0.00),v40,z0,tPen\WObj:=wPaper;
    MoveL Offs(pOrigin,158.68,93.90,0.00),v40,z0,tPen\WObj:=wPaper;
    MoveL Offs(pOrigin,153.26,95.70,0.00),v40,z0,tPen\WObj:=wPaper;
    MoveL Offs(pOrigin,151.46,96.69,0.00),v40,fine,tPen\WObj:=wPaper;
    MoveL Offs(pOrigin,151.46,96.69,6.00),v60,z5,tPen\WObj:=wPaper;
    MoveL Offs(pOrigin,146.14,100.09,6.00),vTravel,z5,tPen\WObj:=wPaper;
    MoveL Offs(pOrigin,146.14,100.09,0.00),v60,z0,tPen\WObj:=wPaper;
    MoveL Offs(pOrigin,145.82,100.41,0.00),v40,z0,tPen\WObj:=wPaper;
    MoveL Offs(pOrigin,146.14,100.09,0.00),v40,fine,tPen\WObj:=wPaper;
    MoveL Offs(pOrigin,146.14,100.09,6.00),v60,z5,tPen\WObj:=wPaper;
    MoveL Offs(pOrigin,143.38,102.01,6.00),vTravel,z5,tPen\WObj:=wPaper;
    MoveL Offs(pOrigin,143.38,102.01,0.00),v60,z0,tPen\WObj:=wPaper;
    MoveL Offs(pOrigin,144.98,101.16,0.00),v40,z0,tPen\WObj:=wPaper;
    MoveL Offs(pOrigin,149.76,97.30,0.00),v40,z0,tPen\WObj:=wPaper;
    MoveL Offs(pOrigin,151.35,96.73,0.00),v40,z0,tPen\WObj:=wPaper;
    MoveL Offs(pOrigin,157.30,99.88,0.00),v40,z0,tPen\WObj:=wPaper;
    MoveL Offs(pOrigin,156.98,100.73,0.00),v40,z0,tPen\WObj:=wPaper;
    MoveL Offs(pOrigin,154.36,104.03,0.00),v40,z0,tPen\WObj:=wPaper;
    MoveL Offs(pOrigin,154.22,104.66,0.00),v40,fine,tPen\WObj:=wPaper;
  ENDPROC

  PROC DrawPart9()
    MoveL Offs(pOrigin,154.22,104.66,6.00),v60,z5,tPen\WObj:=wPaper;
    MoveL Offs(pOrigin,152.84,105.94,6.00),vTravel,z5,tPen\WObj:=wPaper;
    MoveL Offs(pOrigin,152.84,105.94,0.00),v60,z0,tPen\WObj:=wPaper;
    MoveL Offs(pOrigin,152.52,106.26,0.00),v40,z0,tPen\WObj:=wPaper;
    MoveL Offs(pOrigin,152.84,105.94,0.00),v40,fine,tPen\WObj:=wPaper;
    MoveL Offs(pOrigin,152.84,105.94,6.00),v60,z5,tPen\WObj:=wPaper;
    MoveL Offs(pOrigin,151.88,107.11,6.00),vTravel,z5,tPen\WObj:=wPaper;
    MoveL Offs(pOrigin,151.88,107.11,0.00),v60,z0,tPen\WObj:=wPaper;
    MoveL Offs(pOrigin,151.56,107.43,0.00),v40,z0,tPen\WObj:=wPaper;
    MoveL Offs(pOrigin,151.88,107.11,0.00),v40,fine,tPen\WObj:=wPaper;
    MoveL Offs(pOrigin,151.88,107.11,6.00),v60,z5,tPen\WObj:=wPaper;
    MoveL Offs(pOrigin,157.73,100.84,6.00),vTravel,z5,tPen\WObj:=wPaper;
    MoveL Offs(pOrigin,157.73,100.84,0.00),v60,z0,tPen\WObj:=wPaper;
    MoveL Offs(pOrigin,159.35,98.18,0.00),v40,z0,tPen\WObj:=wPaper;
    MoveL Offs(pOrigin,160.27,95.31,0.00),v40,z0,tPen\WObj:=wPaper;
    MoveL Offs(pOrigin,160.27,92.12,0.00),v40,z0,tPen\WObj:=wPaper;
    MoveL Offs(pOrigin,159.32,88.51,0.00),v40,fine,tPen\WObj:=wPaper;
    MoveL Offs(pOrigin,159.32,88.51,6.00),v60,z5,tPen\WObj:=wPaper;
    MoveL Offs(pOrigin,165.52,88.80,6.00),vTravel,z5,tPen\WObj:=wPaper;
    MoveL Offs(pOrigin,165.52,88.80,0.00),v60,z0,tPen\WObj:=wPaper;
    MoveL Offs(pOrigin,166.86,90.11,0.00),v40,z0,tPen\WObj:=wPaper;
    MoveL Offs(pOrigin,165.52,88.80,0.00),v40,fine,tPen\WObj:=wPaper;
    MoveL Offs(pOrigin,165.52,88.80,6.00),v60,z5,tPen\WObj:=wPaper;
    MoveL Offs(pOrigin,170.16,92.97,6.00),vTravel,z5,tPen\WObj:=wPaper;
    MoveL Offs(pOrigin,170.16,92.97,0.00),v60,z0,tPen\WObj:=wPaper;
    MoveL Offs(pOrigin,165.38,88.72,0.00),v40,z0,tPen\WObj:=wPaper;
    MoveL Offs(pOrigin,161.87,84.58,0.00),v40,z0,tPen\WObj:=wPaper;
    MoveL Offs(pOrigin,157.48,78.10,0.00),v40,z0,tPen\WObj:=wPaper;
    MoveL Offs(pOrigin,155.07,73.43,0.00),v40,fine,tPen\WObj:=wPaper;
    MoveL Offs(pOrigin,155.07,73.43,6.00),v60,z5,tPen\WObj:=wPaper;
    MoveL Offs(pOrigin,152.73,87.03,6.00),vTravel,z5,tPen\WObj:=wPaper;
    MoveL Offs(pOrigin,152.73,87.03,0.00),v60,z0,tPen\WObj:=wPaper;
    MoveL Offs(pOrigin,148.69,88.58,0.00),v40,z0,tPen\WObj:=wPaper;
    MoveL Offs(pOrigin,148.41,89.01,0.00),v40,z0,tPen\WObj:=wPaper;
    MoveL Offs(pOrigin,152.09,87.91,0.00),v40,z0,tPen\WObj:=wPaper;
    MoveL Offs(pOrigin,153.01,87.24,0.00),v40,z0,tPen\WObj:=wPaper;
    MoveL Offs(pOrigin,152.73,87.03,0.00),v40,fine,tPen\WObj:=wPaper;
    MoveL Offs(pOrigin,152.73,87.03,6.00),v60,z5,tPen\WObj:=wPaper;
    MoveL Offs(pOrigin,140.19,90.43,6.00),vTravel,z5,tPen\WObj:=wPaper;
    MoveL Offs(pOrigin,140.19,90.43,0.00),v60,z0,tPen\WObj:=wPaper;
    MoveL Offs(pOrigin,139.73,90.74,0.00),v40,z0,tPen\WObj:=wPaper;
    MoveL Offs(pOrigin,138.92,93.29,0.00),v40,z0,tPen\WObj:=wPaper;
    MoveL Offs(pOrigin,138.92,93.29,0.00),v40,z0,tPen\WObj:=wPaper;
    MoveL Offs(pOrigin,138.71,94.99,0.00),v40,z0,tPen\WObj:=wPaper;
    MoveL Offs(pOrigin,137.96,96.48,0.00),v40,z0,tPen\WObj:=wPaper;
    MoveL Offs(pOrigin,137.75,96.59,0.00),v40,z0,tPen\WObj:=wPaper;
    MoveL Offs(pOrigin,137.01,96.80,0.00),v40,z0,tPen\WObj:=wPaper;
    MoveL Offs(pOrigin,136.16,96.27,0.00),v40,z0,tPen\WObj:=wPaper;
    MoveL Offs(pOrigin,133.50,91.91,0.00),v40,fine,tPen\WObj:=wPaper;
    MoveL Offs(pOrigin,133.50,91.91,6.00),v60,z5,tPen\WObj:=wPaper;
    MoveL Offs(pOrigin,134.03,90.53,6.00),vTravel,z5,tPen\WObj:=wPaper;
    MoveL Offs(pOrigin,134.03,90.53,0.00),v60,z0,tPen\WObj:=wPaper;
    MoveL Offs(pOrigin,138.92,93.29,0.00),v40,fine,tPen\WObj:=wPaper;
    MoveL Offs(pOrigin,138.92,93.29,6.00),v60,z5,tPen\WObj:=wPaper;
    MoveL Offs(pOrigin,138.81,91.59,6.00),vTravel,z5,tPen\WObj:=wPaper;
    MoveL Offs(pOrigin,138.81,91.59,0.00),v60,z0,tPen\WObj:=wPaper;
    MoveL Offs(pOrigin,134.99,82.78,0.00),v40,fine,tPen\WObj:=wPaper;
    MoveL Offs(pOrigin,134.99,82.78,6.00),v60,z5,tPen\WObj:=wPaper;
    MoveL Offs(pOrigin,137.86,78.84,6.00),vTravel,z5,tPen\WObj:=wPaper;
    MoveL Offs(pOrigin,137.86,78.84,0.00),v60,z0,tPen\WObj:=wPaper;
    MoveL Offs(pOrigin,137.25,78.42,0.00),v40,z0,tPen\WObj:=wPaper;
    MoveL Offs(pOrigin,134.35,71.09,0.00),v40,fine,tPen\WObj:=wPaper;
    MoveL Offs(pOrigin,134.35,71.09,6.00),v60,z5,tPen\WObj:=wPaper;
    MoveL Offs(pOrigin,127.90,78.21,6.00),vTravel,z5,tPen\WObj:=wPaper;
    MoveL Offs(pOrigin,127.90,78.21,0.00),v60,z0,tPen\WObj:=wPaper;
    MoveL Offs(pOrigin,126.81,77.46,0.00),v40,z0,tPen\WObj:=wPaper;
    MoveL Offs(pOrigin,126.06,77.64,0.00),v40,z0,tPen\WObj:=wPaper;
    MoveL Offs(pOrigin,125.39,78.31,0.00),v40,z0,tPen\WObj:=wPaper;
    MoveL Offs(pOrigin,125.39,79.59,0.00),v40,z0,tPen\WObj:=wPaper;
    MoveL Offs(pOrigin,126.59,80.44,0.00),v40,z0,tPen\WObj:=wPaper;
    MoveL Offs(pOrigin,127.44,80.15,0.00),v40,z0,tPen\WObj:=wPaper;
    MoveL Offs(pOrigin,128.08,79.06,0.00),v40,z0,tPen\WObj:=wPaper;
    MoveL Offs(pOrigin,127.90,78.21,0.00),v40,fine,tPen\WObj:=wPaper;
    MoveL Offs(pOrigin,127.90,78.21,6.00),v60,z5,tPen\WObj:=wPaper;
    MoveL Offs(pOrigin,125.43,79.48,6.00),vTravel,z5,tPen\WObj:=wPaper;
    MoveL Offs(pOrigin,125.43,79.48,0.00),v60,z0,tPen\WObj:=wPaper;
    MoveL Offs(pOrigin,125.96,80.12,0.00),v40,z0,tPen\WObj:=wPaper;
    MoveL Offs(pOrigin,125.43,79.48,0.00),v40,fine,tPen\WObj:=wPaper;
    MoveL Offs(pOrigin,125.43,79.48,6.00),v60,z5,tPen\WObj:=wPaper;
    MoveL Offs(pOrigin,126.49,84.37,6.00),vTravel,z5,tPen\WObj:=wPaper;
    MoveL Offs(pOrigin,126.49,84.37,0.00),v60,z0,tPen\WObj:=wPaper;
    MoveL Offs(pOrigin,128.51,85.96,0.00),v40,z0,tPen\WObj:=wPaper;
    MoveL Offs(pOrigin,129.71,87.45,0.00),v40,z0,tPen\WObj:=wPaper;
    MoveL Offs(pOrigin,130.60,90.43,0.00),v40,z0,tPen\WObj:=wPaper;
    MoveL Offs(pOrigin,134.77,96.91,0.00),v40,z0,tPen\WObj:=wPaper;
    MoveL Offs(pOrigin,134.77,96.91,0.00),v40,z0,tPen\WObj:=wPaper;
    MoveL Offs(pOrigin,137.25,100.31,0.00),v40,z0,tPen\WObj:=wPaper;
    MoveL Offs(pOrigin,140.19,105.83,0.00),v40,fine,tPen\WObj:=wPaper;
    MoveL Offs(pOrigin,140.19,105.83,6.00),v60,z5,tPen\WObj:=wPaper;
    MoveL Offs(pOrigin,137.64,101.37,6.00),vTravel,z5,tPen\WObj:=wPaper;
    MoveL Offs(pOrigin,137.64,101.37,0.00),v60,z0,tPen\WObj:=wPaper;
    MoveL Offs(pOrigin,133.29,99.00,0.00),v40,z0,tPen\WObj:=wPaper;
    MoveL Offs(pOrigin,131.27,98.29,0.00),v40,z0,tPen\WObj:=wPaper;
    MoveL Offs(pOrigin,129.04,97.97,0.00),v40,z0,tPen\WObj:=wPaper;
    MoveL Offs(pOrigin,126.59,98.39,0.00),v40,fine,tPen\WObj:=wPaper;
    MoveL Offs(pOrigin,126.59,98.39,6.00),v60,z5,tPen\WObj:=wPaper;
    MoveL Offs(pOrigin,122.34,97.97,6.00),vTravel,z5,tPen\WObj:=wPaper;
    MoveL Offs(pOrigin,122.34,97.97,0.00),v60,z0,tPen\WObj:=wPaper;
    MoveL Offs(pOrigin,119.26,98.68,0.00),v40,z0,tPen\WObj:=wPaper;
    MoveL Offs(pOrigin,115.86,100.41,0.00),v40,z0,tPen\WObj:=wPaper;
    MoveL Offs(pOrigin,114.23,102.64,0.00),v40,z0,tPen\WObj:=wPaper;
    MoveL Offs(pOrigin,113.53,104.34,0.00),v40,fine,tPen\WObj:=wPaper;
    MoveL Offs(pOrigin,113.53,104.34,6.00),v60,z5,tPen\WObj:=wPaper;
    MoveL Offs(pOrigin,111.19,100.41,6.00),vTravel,z5,tPen\WObj:=wPaper;
    MoveL Offs(pOrigin,111.19,100.41,0.00),v60,z0,tPen\WObj:=wPaper;
    MoveL Offs(pOrigin,110.34,99.99,0.00),v40,z0,tPen\WObj:=wPaper;
    MoveL Offs(pOrigin,106.62,96.59,0.00),v40,z0,tPen\WObj:=wPaper;
    MoveL Offs(pOrigin,104.39,95.21,0.00),v40,z0,tPen\WObj:=wPaper;
    MoveL Offs(pOrigin,98.86,97.12,0.00),v40,z0,tPen\WObj:=wPaper;
    MoveL Offs(pOrigin,98.97,97.86,0.00),v40,z0,tPen\WObj:=wPaper;
    MoveL Offs(pOrigin,105.13,105.09,0.00),v40,z0,tPen\WObj:=wPaper;
    MoveL Offs(pOrigin,105.34,105.94,0.00),v40,z0,tPen\WObj:=wPaper;
    MoveL Offs(pOrigin,105.34,105.94,0.00),v40,z0,tPen\WObj:=wPaper;
    MoveL Offs(pOrigin,107.89,108.17,0.00),v40,z0,tPen\WObj:=wPaper;
    MoveL Offs(pOrigin,108.21,108.91,0.00),v40,z0,tPen\WObj:=wPaper;
    MoveL Offs(pOrigin,108.21,108.91,0.00),v40,z0,tPen\WObj:=wPaper;
    MoveL Offs(pOrigin,104.28,108.59,0.00),v40,z0,tPen\WObj:=wPaper;
    MoveL Offs(pOrigin,100.56,107.57,0.00),v40,z0,tPen\WObj:=wPaper;
    MoveL Offs(pOrigin,90.47,102.61,0.00),v40,z0,tPen\WObj:=wPaper;
    MoveL Offs(pOrigin,86.86,101.16,0.00),v40,z0,tPen\WObj:=wPaper;
  ENDPROC

  PROC DrawPart10()
    MoveL Offs(pOrigin,86.01,101.16,0.00),v40,z0,tPen\WObj:=wPaper;
    MoveL Offs(pOrigin,85.16,103.81,0.00),v40,z0,tPen\WObj:=wPaper;
    MoveL Offs(pOrigin,84.41,107.96,0.00),v40,z0,tPen\WObj:=wPaper;
    MoveL Offs(pOrigin,84.41,110.93,0.00),v40,z0,tPen\WObj:=wPaper;
    MoveL Offs(pOrigin,85.01,113.91,0.00),v40,z0,tPen\WObj:=wPaper;
    MoveL Offs(pOrigin,86.11,116.03,0.00),v40,z0,tPen\WObj:=wPaper;
    MoveL Offs(pOrigin,87.71,117.62,0.00),v40,z0,tPen\WObj:=wPaper;
    MoveL Offs(pOrigin,90.15,118.94,0.00),v40,z0,tPen\WObj:=wPaper;
    MoveL Offs(pOrigin,93.02,119.64,0.00),v40,fine,tPen\WObj:=wPaper;
    MoveL Offs(pOrigin,93.02,119.64,6.00),v60,z5,tPen\WObj:=wPaper;
    MoveL Offs(pOrigin,85.26,116.99,6.00),vTravel,z5,tPen\WObj:=wPaper;
    MoveL Offs(pOrigin,85.26,116.99,0.00),v60,z0,tPen\WObj:=wPaper;
    MoveL Offs(pOrigin,83.85,114.86,0.00),v40,z0,tPen\WObj:=wPaper;
    MoveL Offs(pOrigin,82.82,111.78,0.00),v40,z0,tPen\WObj:=wPaper;
    MoveL Offs(pOrigin,82.61,106.36,0.00),v40,z0,tPen\WObj:=wPaper;
    MoveL Offs(pOrigin,83.70,100.31,0.00),v40,z0,tPen\WObj:=wPaper;
    MoveL Offs(pOrigin,84.52,100.31,0.00),v40,z0,tPen\WObj:=wPaper;
    MoveL Offs(pOrigin,86.01,101.05,0.00),v40,fine,tPen\WObj:=wPaper;
    MoveL Offs(pOrigin,86.01,101.05,6.00),v60,z5,tPen\WObj:=wPaper;
    MoveL Offs(pOrigin,83.67,100.20,6.00),vTravel,z5,tPen\WObj:=wPaper;
    MoveL Offs(pOrigin,83.67,100.20,0.00),v60,z0,tPen\WObj:=wPaper;
    MoveL Offs(pOrigin,80.16,99.14,0.00),v40,fine,tPen\WObj:=wPaper;
    MoveL Offs(pOrigin,80.16,99.14,6.00),v60,z5,tPen\WObj:=wPaper;
    MoveL Offs(pOrigin,79.95,97.54,6.00),vTravel,z5,tPen\WObj:=wPaper;
    MoveL Offs(pOrigin,79.95,97.54,0.00),v60,z0,tPen\WObj:=wPaper;
    MoveL Offs(pOrigin,89.72,100.59,0.00),v40,z0,tPen\WObj:=wPaper;
    MoveL Offs(pOrigin,97.16,104.17,0.00),v40,z0,tPen\WObj:=wPaper;
    MoveL Offs(pOrigin,99.50,104.98,0.00),v40,z0,tPen\WObj:=wPaper;
    MoveL Offs(pOrigin,105.34,105.94,0.00),v40,fine,tPen\WObj:=wPaper;
    MoveL Offs(pOrigin,105.34,105.94,6.00),v60,z5,tPen\WObj:=wPaper;
    MoveL Offs(pOrigin,106.76,106.96,6.00),vTravel,z5,tPen\WObj:=wPaper;
    MoveL Offs(pOrigin,106.76,106.96,0.00),v60,z0,tPen\WObj:=wPaper;
    MoveL Offs(pOrigin,107.79,107.96,0.00),v40,z0,tPen\WObj:=wPaper;
    MoveL Offs(pOrigin,106.76,106.96,0.00),v40,fine,tPen\WObj:=wPaper;
    MoveL Offs(pOrigin,106.76,106.96,6.00),v60,z5,tPen\WObj:=wPaper;
    MoveL Offs(pOrigin,100.46,101.79,6.00),vTravel,z5,tPen\WObj:=wPaper;
    MoveL Offs(pOrigin,100.46,101.79,0.00),v60,z0,tPen\WObj:=wPaper;
    MoveL Offs(pOrigin,98.33,99.88,0.00),v40,z0,tPen\WObj:=wPaper;
    MoveL Offs(pOrigin,95.64,96.16,0.00),v40,z0,tPen\WObj:=wPaper;
    MoveL Offs(pOrigin,94.82,93.93,0.00),v40,z0,tPen\WObj:=wPaper;
    MoveL Offs(pOrigin,94.29,91.06,0.00),v40,z0,tPen\WObj:=wPaper;
    MoveL Offs(pOrigin,94.72,83.62,0.00),v40,fine,tPen\WObj:=wPaper;
    MoveL Offs(pOrigin,94.72,83.62,6.00),v60,z5,tPen\WObj:=wPaper;
    MoveL Offs(pOrigin,91.96,77.04,6.00),vTravel,z5,tPen\WObj:=wPaper;
    MoveL Offs(pOrigin,91.96,77.04,0.00),v60,z0,tPen\WObj:=wPaper;
    MoveL Offs(pOrigin,91.32,72.26,0.00),v40,z0,tPen\WObj:=wPaper;
    MoveL Offs(pOrigin,89.76,67.58,0.00),v40,z0,tPen\WObj:=wPaper;
    MoveL Offs(pOrigin,87.64,63.54,0.00),v40,z0,tPen\WObj:=wPaper;
    MoveL Offs(pOrigin,81.44,54.09,0.00),v40,z0,tPen\WObj:=wPaper;
    MoveL Offs(pOrigin,81.44,54.09,0.00),v40,z0,tPen\WObj:=wPaper;
    MoveL Offs(pOrigin,78.25,55.61,0.00),v40,z0,tPen\WObj:=wPaper;
    MoveL Offs(pOrigin,75.38,56.42,0.00),v40,fine,tPen\WObj:=wPaper;
    MoveL Offs(pOrigin,75.38,56.42,6.00),v60,z5,tPen\WObj:=wPaper;
    MoveL Offs(pOrigin,71.98,60.04,6.00),vTravel,z5,tPen\WObj:=wPaper;
    MoveL Offs(pOrigin,71.98,60.04,0.00),v60,z0,tPen\WObj:=wPaper;
    MoveL Offs(pOrigin,76.02,60.89,0.00),v40,z0,tPen\WObj:=wPaper;
    MoveL Offs(pOrigin,77.82,60.78,0.00),v40,z0,tPen\WObj:=wPaper;
    MoveL Offs(pOrigin,79.42,60.14,0.00),v40,z0,tPen\WObj:=wPaper;
    MoveL Offs(pOrigin,79.74,60.04,0.00),v40,z0,tPen\WObj:=wPaper;
    MoveL Offs(pOrigin,80.59,59.72,0.00),v40,z0,tPen\WObj:=wPaper;
    MoveL Offs(pOrigin,80.59,59.72,0.00),v40,z0,tPen\WObj:=wPaper;
    MoveL Offs(pOrigin,79.95,64.50,0.00),v40,z0,tPen\WObj:=wPaper;
    MoveL Offs(pOrigin,79.95,64.50,0.00),v40,z0,tPen\WObj:=wPaper;
    MoveL Offs(pOrigin,79.53,66.73,0.00),v40,z0,tPen\WObj:=wPaper;
    MoveL Offs(pOrigin,79.53,66.73,0.00),v40,z0,tPen\WObj:=wPaper;
    MoveL Offs(pOrigin,79.21,68.86,0.00),v40,z0,tPen\WObj:=wPaper;
    MoveL Offs(pOrigin,78.57,70.24,0.00),v40,z0,tPen\WObj:=wPaper;
    MoveL Offs(pOrigin,77.82,70.34,0.00),v40,z0,tPen\WObj:=wPaper;
    MoveL Offs(pOrigin,77.47,71.30,0.00),v40,z0,tPen\WObj:=wPaper;
    MoveL Offs(pOrigin,74.18,75.12,0.00),v40,z0,tPen\WObj:=wPaper;
    MoveL Offs(pOrigin,70.49,78.53,0.00),v40,z0,tPen\WObj:=wPaper;
    MoveL Offs(pOrigin,70.28,78.63,0.00),v40,z0,tPen\WObj:=wPaper;
    MoveL Offs(pOrigin,67.52,80.01,0.00),v40,fine,tPen\WObj:=wPaper;
    MoveL Offs(pOrigin,67.52,80.01,6.00),v60,z5,tPen\WObj:=wPaper;
    MoveL Offs(pOrigin,70.39,74.81,6.00),vTravel,z5,tPen\WObj:=wPaper;
    MoveL Offs(pOrigin,70.39,74.81,0.00),v60,z0,tPen\WObj:=wPaper;
    MoveL Offs(pOrigin,73.26,73.32,0.00),v40,z0,tPen\WObj:=wPaper;
    MoveL Offs(pOrigin,73.57,73.21,0.00),v40,z0,tPen\WObj:=wPaper;
    MoveL Offs(pOrigin,77.08,70.56,0.00),v40,z0,tPen\WObj:=wPaper;
    MoveL Offs(pOrigin,77.82,70.34,0.00),v40,z0,tPen\WObj:=wPaper;
    MoveL Offs(pOrigin,77.82,70.34,0.00),v40,z0,tPen\WObj:=wPaper;
    MoveL Offs(pOrigin,78.57,70.34,0.00),v40,z0,tPen\WObj:=wPaper;
    MoveL Offs(pOrigin,78.68,71.09,0.00),v40,z0,tPen\WObj:=wPaper;
    MoveL Offs(pOrigin,75.06,82.14,0.00),v40,fine,tPen\WObj:=wPaper;
    MoveL Offs(pOrigin,75.06,82.14,6.00),v60,z5,tPen\WObj:=wPaper;
    MoveL Offs(pOrigin,74.85,77.78,6.00),vTravel,z5,tPen\WObj:=wPaper;
    MoveL Offs(pOrigin,74.85,77.78,0.00),v60,z0,tPen\WObj:=wPaper;
    MoveL Offs(pOrigin,70.32,82.24,0.00),v40,z0,tPen\WObj:=wPaper;
    MoveL Offs(pOrigin,67.62,86.28,0.00),v40,fine,tPen\WObj:=wPaper;
    MoveL Offs(pOrigin,67.62,86.28,6.00),v60,z5,tPen\WObj:=wPaper;
    MoveL Offs(pOrigin,71.56,88.30,6.00),vTravel,z5,tPen\WObj:=wPaper;
    MoveL Offs(pOrigin,71.56,88.30,0.00),v60,z0,tPen\WObj:=wPaper;
    MoveL Offs(pOrigin,74.43,82.46,0.00),v40,z0,tPen\WObj:=wPaper;
    MoveL Offs(pOrigin,74.96,82.17,0.00),v40,z0,tPen\WObj:=wPaper;
    MoveL Offs(pOrigin,75.06,82.78,0.00),v40,z0,tPen\WObj:=wPaper;
    MoveL Offs(pOrigin,72.62,91.59,0.00),v40,z0,tPen\WObj:=wPaper;
    MoveL Offs(pOrigin,72.51,96.38,0.00),v40,fine,tPen\WObj:=wPaper;
    MoveL Offs(pOrigin,72.51,96.38,6.00),v60,z5,tPen\WObj:=wPaper;
    MoveL Offs(pOrigin,87.07,89.04,6.00),vTravel,z5,tPen\WObj:=wPaper;
    MoveL Offs(pOrigin,87.07,89.04,0.00),v60,z0,tPen\WObj:=wPaper;
    MoveL Offs(pOrigin,88.17,87.34,0.00),v40,z0,tPen\WObj:=wPaper;
    MoveL Offs(pOrigin,89.19,84.58,0.00),v40,z0,tPen\WObj:=wPaper;
    MoveL Offs(pOrigin,89.62,79.16,0.00),v40,z0,tPen\WObj:=wPaper;
    MoveL Offs(pOrigin,88.56,73.21,0.00),v40,z0,tPen\WObj:=wPaper;
    MoveL Offs(pOrigin,86.11,67.26,0.00),v40,fine,tPen\WObj:=wPaper;
    MoveL Offs(pOrigin,86.11,67.26,6.00),v60,z5,tPen\WObj:=wPaper;
    MoveL Offs(pOrigin,85.90,63.86,6.00),vTravel,z5,tPen\WObj:=wPaper;
    MoveL Offs(pOrigin,85.90,63.86,0.00),v60,z0,tPen\WObj:=wPaper;
    MoveL Offs(pOrigin,81.37,56.53,0.00),v40,z0,tPen\WObj:=wPaper;
    MoveL Offs(pOrigin,81.54,54.62,0.00),v40,fine,tPen\WObj:=wPaper;
    MoveL Offs(pOrigin,81.54,54.62,6.00),v60,z5,tPen\WObj:=wPaper;
    MoveL Offs(pOrigin,81.33,56.64,6.00),vTravel,z5,tPen\WObj:=wPaper;
    MoveL Offs(pOrigin,81.33,56.64,0.00),v60,z0,tPen\WObj:=wPaper;
    MoveL Offs(pOrigin,80.59,59.72,0.00),v40,fine,tPen\WObj:=wPaper;
    MoveL Offs(pOrigin,80.59,59.72,6.00),v60,z5,tPen\WObj:=wPaper;
    MoveL Offs(pOrigin,80.91,57.91,6.00),vTravel,z5,tPen\WObj:=wPaper;
    MoveL Offs(pOrigin,80.91,57.91,0.00),v60,z0,tPen\WObj:=wPaper;
    MoveL Offs(pOrigin,78.04,57.91,0.00),v40,z0,tPen\WObj:=wPaper;
    MoveL Offs(pOrigin,70.81,58.66,0.00),v40,z0,tPen\WObj:=wPaper;
    MoveL Offs(pOrigin,65.71,58.55,0.00),v40,z0,tPen\WObj:=wPaper;
  ENDPROC

  PROC DrawPart11()
    MoveL Offs(pOrigin,62.95,58.12,0.00),v40,fine,tPen\WObj:=wPaper;
    MoveL Offs(pOrigin,62.95,58.12,6.00),v60,z5,tPen\WObj:=wPaper;
    MoveL Offs(pOrigin,63.48,59.72,6.00),vTravel,z5,tPen\WObj:=wPaper;
    MoveL Offs(pOrigin,63.48,59.72,0.00),v60,z0,tPen\WObj:=wPaper;
    MoveL Offs(pOrigin,59.66,58.59,0.00),v40,z0,tPen\WObj:=wPaper;
    MoveL Offs(pOrigin,57.21,57.17,0.00),v40,z0,tPen\WObj:=wPaper;
    MoveL Offs(pOrigin,55.41,55.26,0.00),v40,z0,tPen\WObj:=wPaper;
    MoveL Offs(pOrigin,53.60,51.96,0.00),v40,fine,tPen\WObj:=wPaper;
    MoveL Offs(pOrigin,53.60,51.96,6.00),v60,z5,tPen\WObj:=wPaper;
    MoveL Offs(pOrigin,52.01,49.84,6.00),vTravel,z5,tPen\WObj:=wPaper;
    MoveL Offs(pOrigin,52.01,49.84,0.00),v60,z0,tPen\WObj:=wPaper;
    MoveL Offs(pOrigin,53.07,50.12,0.00),v40,z0,tPen\WObj:=wPaper;
    MoveL Offs(pOrigin,59.55,53.88,0.00),v40,fine,tPen\WObj:=wPaper;
    MoveL Offs(pOrigin,59.55,53.88,6.00),v60,z5,tPen\WObj:=wPaper;
    MoveL Offs(pOrigin,56.04,56.00,6.00),vTravel,z5,tPen\WObj:=wPaper;
    MoveL Offs(pOrigin,56.04,56.00,0.00),v60,z0,tPen\WObj:=wPaper;
    MoveL Offs(pOrigin,56.47,56.42,0.00),v40,z0,tPen\WObj:=wPaper;
    MoveL Offs(pOrigin,56.04,56.00,0.00),v40,fine,tPen\WObj:=wPaper;
    MoveL Offs(pOrigin,56.04,56.00,6.00),v60,z5,tPen\WObj:=wPaper;
    MoveL Offs(pOrigin,58.70,59.83,6.00),vTravel,z5,tPen\WObj:=wPaper;
    MoveL Offs(pOrigin,58.70,59.83,0.00),v60,z0,tPen\WObj:=wPaper;
    MoveL Offs(pOrigin,63.80,62.76,0.00),v40,z0,tPen\WObj:=wPaper;
    MoveL Offs(pOrigin,65.82,64.50,0.00),v40,fine,tPen\WObj:=wPaper;
    MoveL Offs(pOrigin,65.82,64.50,6.00),v60,z5,tPen\WObj:=wPaper;
    MoveL Offs(pOrigin,69.32,60.78,6.00),vTravel,z5,tPen\WObj:=wPaper;
    MoveL Offs(pOrigin,69.32,60.78,0.00),v60,z0,tPen\WObj:=wPaper;
    MoveL Offs(pOrigin,74.53,62.27,0.00),v40,z0,tPen\WObj:=wPaper;
    MoveL Offs(pOrigin,78.68,62.38,0.00),v40,fine,tPen\WObj:=wPaper;
    MoveL Offs(pOrigin,78.68,62.38,6.00),v60,z5,tPen\WObj:=wPaper;
    MoveL Offs(pOrigin,79.95,64.50,6.00),vTravel,z5,tPen\WObj:=wPaper;
    MoveL Offs(pOrigin,79.95,64.50,0.00),v60,z0,tPen\WObj:=wPaper;
    MoveL Offs(pOrigin,79.31,64.64,0.00),v40,z0,tPen\WObj:=wPaper;
    MoveL Offs(pOrigin,76.87,66.55,0.00),v40,z0,tPen\WObj:=wPaper;
    MoveL Offs(pOrigin,74.32,67.94,0.00),v40,z0,tPen\WObj:=wPaper;
    MoveL Offs(pOrigin,70.28,69.28,0.00),v40,fine,tPen\WObj:=wPaper;
    MoveL Offs(pOrigin,70.28,69.28,6.00),v60,z5,tPen\WObj:=wPaper;
    MoveL Offs(pOrigin,67.73,71.41,6.00),vTravel,z5,tPen\WObj:=wPaper;
    MoveL Offs(pOrigin,67.73,71.41,0.00),v60,z0,tPen\WObj:=wPaper;
    MoveL Offs(pOrigin,70.60,71.09,0.00),v40,z0,tPen\WObj:=wPaper;
    MoveL Offs(pOrigin,73.68,70.17,0.00),v40,z0,tPen\WObj:=wPaper;
    MoveL Offs(pOrigin,77.72,67.90,0.00),v40,z0,tPen\WObj:=wPaper;
    MoveL Offs(pOrigin,77.93,67.79,0.00),v40,z0,tPen\WObj:=wPaper;
    MoveL Offs(pOrigin,79.53,66.73,0.00),v40,fine,tPen\WObj:=wPaper;
    MoveL Offs(pOrigin,79.53,66.73,6.00),v60,z5,tPen\WObj:=wPaper;
    MoveL Offs(pOrigin,74.74,65.88,6.00),vTravel,z5,tPen\WObj:=wPaper;
    MoveL Offs(pOrigin,74.74,65.88,0.00),v60,z0,tPen\WObj:=wPaper;
    MoveL Offs(pOrigin,68.37,68.01,0.00),v40,z0,tPen\WObj:=wPaper;
    MoveL Offs(pOrigin,61.89,69.07,0.00),v40,fine,tPen\WObj:=wPaper;
    MoveL Offs(pOrigin,61.89,69.07,6.00),v60,z5,tPen\WObj:=wPaper;
    MoveL Offs(pOrigin,66.56,50.58,6.00),vTravel,z5,tPen\WObj:=wPaper;
    MoveL Offs(pOrigin,66.56,50.58,0.00),v60,z0,tPen\WObj:=wPaper;
    MoveL Offs(pOrigin,69.22,50.16,0.00),v40,z0,tPen\WObj:=wPaper;
    MoveL Offs(pOrigin,72.94,48.49,0.00),v40,z0,tPen\WObj:=wPaper;
    MoveL Offs(pOrigin,76.23,45.80,0.00),v40,z0,tPen\WObj:=wPaper;
    MoveL Offs(pOrigin,78.57,42.61,0.00),v40,fine,tPen\WObj:=wPaper;
    MoveL Offs(pOrigin,78.57,42.61,6.00),v60,z5,tPen\WObj:=wPaper;
    MoveL Offs(pOrigin,79.42,41.12,6.00),vTravel,z5,tPen\WObj:=wPaper;
    MoveL Offs(pOrigin,79.42,41.12,0.00),v60,z0,tPen\WObj:=wPaper;
    MoveL Offs(pOrigin,84.52,39.21,0.00),v40,z0,tPen\WObj:=wPaper;
    MoveL Offs(pOrigin,84.52,39.21,0.00),v40,z0,tPen\WObj:=wPaper;
    MoveL Offs(pOrigin,81.22,49.31,0.00),v40,z0,tPen\WObj:=wPaper;
    MoveL Offs(pOrigin,80.48,48.67,0.00),v40,z0,tPen\WObj:=wPaper;
    MoveL Offs(pOrigin,81.19,49.41,0.00),v40,z0,tPen\WObj:=wPaper;
    MoveL Offs(pOrigin,81.76,51.01,0.00),v40,fine,tPen\WObj:=wPaper;
    MoveL Offs(pOrigin,81.76,51.01,6.00),v60,z5,tPen\WObj:=wPaper;
    MoveL Offs(pOrigin,82.82,50.26,6.00),vTravel,z5,tPen\WObj:=wPaper;
    MoveL Offs(pOrigin,82.82,50.26,0.00),v60,z0,tPen\WObj:=wPaper;
    MoveL Offs(pOrigin,83.99,51.11,0.00),v40,z0,tPen\WObj:=wPaper;
    MoveL Offs(pOrigin,84.84,50.79,0.00),v40,z0,tPen\WObj:=wPaper;
    MoveL Offs(pOrigin,84.73,50.47,0.00),v40,z0,tPen\WObj:=wPaper;
    MoveL Offs(pOrigin,92.06,44.21,0.00),v40,z0,tPen\WObj:=wPaper;
    MoveL Offs(pOrigin,92.28,44.10,0.00),v40,z0,tPen\WObj:=wPaper;
    MoveL Offs(pOrigin,93.76,42.72,0.00),v40,z0,tPen\WObj:=wPaper;
    MoveL Offs(pOrigin,93.76,42.72,0.00),v40,z0,tPen\WObj:=wPaper;
    MoveL Offs(pOrigin,94.61,41.87,0.00),v40,z0,tPen\WObj:=wPaper;
    MoveL Offs(pOrigin,94.61,41.66,0.00),v40,z0,tPen\WObj:=wPaper;
    MoveL Offs(pOrigin,96.03,40.38,0.00),v40,z0,tPen\WObj:=wPaper;
    MoveL Offs(pOrigin,96.10,39.85,0.00),v40,z0,tPen\WObj:=wPaper;
    MoveL Offs(pOrigin,96.10,39.85,0.00),v40,z0,tPen\WObj:=wPaper;
    MoveL Offs(pOrigin,98.12,38.89,0.00),v40,z0,tPen\WObj:=wPaper;
    MoveL Offs(pOrigin,98.30,39.11,0.00),v40,z0,tPen\WObj:=wPaper;
    MoveL Offs(pOrigin,97.80,40.28,0.00),v40,z0,tPen\WObj:=wPaper;
    MoveL Offs(pOrigin,97.80,40.28,0.00),v40,z0,tPen\WObj:=wPaper;
    MoveL Offs(pOrigin,102.16,40.17,0.00),v40,z0,tPen\WObj:=wPaper;
    MoveL Offs(pOrigin,106.19,38.93,0.00),v40,z0,tPen\WObj:=wPaper;
    MoveL Offs(pOrigin,107.29,37.72,0.00),v40,z0,tPen\WObj:=wPaper;
    MoveL Offs(pOrigin,107.57,34.54,0.00),v40,z0,tPen\WObj:=wPaper;
    MoveL Offs(pOrigin,108.00,33.90,0.00),v40,z0,tPen\WObj:=wPaper;
    MoveL Offs(pOrigin,108.00,33.90,0.00),v40,z0,tPen\WObj:=wPaper;
    MoveL Offs(pOrigin,108.43,34.22,0.00),v40,z0,tPen\WObj:=wPaper;
    MoveL Offs(pOrigin,108.74,38.47,0.00),v40,z0,tPen\WObj:=wPaper;
    MoveL Offs(pOrigin,108.21,47.92,0.00),v40,z0,tPen\WObj:=wPaper;
    MoveL Offs(pOrigin,105.88,59.19,0.00),v40,z0,tPen\WObj:=wPaper;
    MoveL Offs(pOrigin,104.46,64.18,0.00),v40,z0,tPen\WObj:=wPaper;
    MoveL Offs(pOrigin,104.07,64.39,0.00),v40,fine,tPen\WObj:=wPaper;
    MoveL Offs(pOrigin,104.07,64.39,6.00),v60,z5,tPen\WObj:=wPaper;
    MoveL Offs(pOrigin,105.24,50.26,6.00),vTravel,z5,tPen\WObj:=wPaper;
    MoveL Offs(pOrigin,105.24,50.26,0.00),v60,z0,tPen\WObj:=wPaper;
    MoveL Offs(pOrigin,103.86,63.33,0.00),v40,z0,tPen\WObj:=wPaper;
    MoveL Offs(pOrigin,104.07,64.93,0.00),v40,z0,tPen\WObj:=wPaper;
    MoveL Offs(pOrigin,97.27,90.74,0.00),v40,z0,tPen\WObj:=wPaper;
    MoveL Offs(pOrigin,97.34,91.28,0.00),v40,z0,tPen\WObj:=wPaper;
    MoveL Offs(pOrigin,103.96,95.10,0.00),v40,fine,tPen\WObj:=wPaper;
    MoveL Offs(pOrigin,103.96,95.10,6.00),v60,z5,tPen\WObj:=wPaper;
    MoveL Offs(pOrigin,107.68,97.44,6.00),vTravel,z5,tPen\WObj:=wPaper;
    MoveL Offs(pOrigin,107.68,97.44,0.00),v60,z0,tPen\WObj:=wPaper;
    MoveL Offs(pOrigin,108.11,97.86,0.00),v40,z0,tPen\WObj:=wPaper;
    MoveL Offs(pOrigin,107.68,97.44,0.00),v40,fine,tPen\WObj:=wPaper;
    MoveL Offs(pOrigin,107.68,97.44,6.00),v60,z5,tPen\WObj:=wPaper;
    MoveL Offs(pOrigin,108.57,98.25,6.00),vTravel,z5,tPen\WObj:=wPaper;
    MoveL Offs(pOrigin,108.57,98.25,0.00),v60,z0,tPen\WObj:=wPaper;
    MoveL Offs(pOrigin,109.49,99.14,0.00),v40,z0,tPen\WObj:=wPaper;
    MoveL Offs(pOrigin,108.57,98.25,0.00),v40,fine,tPen\WObj:=wPaper;
    MoveL Offs(pOrigin,108.57,98.25,6.00),v60,z5,tPen\WObj:=wPaper;
    MoveL Offs(pOrigin,115.86,100.31,6.00),vTravel,z5,tPen\WObj:=wPaper;
    MoveL Offs(pOrigin,115.86,100.31,0.00),v60,z0,tPen\WObj:=wPaper;
    MoveL Offs(pOrigin,117.46,97.65,0.00),v40,z0,tPen\WObj:=wPaper;
    MoveL Offs(pOrigin,119.05,95.95,0.00),v40,fine,tPen\WObj:=wPaper;
    MoveL Offs(pOrigin,119.05,95.95,6.00),v60,z5,tPen\WObj:=wPaper;
    MoveL Offs(pOrigin,114.48,92.02,6.00),vTravel,z5,tPen\WObj:=wPaper;
  ENDPROC

